C07321=1117.098,350.996,-84.045,-177.253,10.967,149.496
C07322=1117.094,351.244,-84.080,-177.250,10.969,149.496
C07323=1117.091,351.491,-84.116,-177.247,10.972,149.496
C07324=1117.087,351.738,-84.151,-177.243,10.974,149.496
C07325=1117.083,351.986,-84.186,-177.240,10.977,149.495
C07326=1117.078,352.233,-84.222,-177.236,10.979,149.495
C07327=1117.075,352.481,-84.258,-177.233,10.981,149.495
C07328=1117.071,352.729,-84.293,-177.230,10.984,149.495
C07329=1117.067,352.976,-84.328,-177.226,10.986,149.494
C07330=1117.063,353.223,-84.364,-177.222,10.989,149.494
C07331=1117.059,353.471,-84.399,-177.219,10.992,149.494
C07332=1117.056,353.718,-84.435,-177.216,10.994,149.494
C07333=1117.052,353.966,-84.470,-177.212,10.996,149.493
C07334=1117.048,354.213,-84.506,-177.209,10.999,149.493
C07335=1117.044,354.460,-84.541,-177.205,11.001,149.493
C07336=1117.040,354.708,-84.576,-177.202,11.004,149.493
C07337=1117.037,354.955,-84.612,-177.199,11.006,149.492
C07338=1117.032,355.203,-84.648,-177.196,11.009,149.492
C07339=1117.029,355.450,-84.684,-177.192,11.011,149.492
C07340=1117.025,355.698,-84.719,-177.188,11.013,149.492
C07341=1117.021,355.945,-84.755,-177.185,11.016,149.491
C07342=1117.017,356.192,-84.790,-177.182,11.018,149.491
C07343=1117.014,356.439,-84.826,-177.179,11.021,149.491
C07344=1117.009,356.687,-84.862,-177.175,11.023,149.491
C07345=1117.006,356.934,-84.898,-177.172,11.025,149.490
C07346=1117.002,357.182,-84.933,-177.168,11.028,149.490
C07347=1116.998,357.429,-84.969,-177.164,11.031,149.490
C07348=1116.995,357.677,-85.005,-177.161,11.033,149.490
C07349=1116.991,357.924,-85.041,-177.158,11.036,149.490
C07350=1116.987,358.172,-85.077,-177.154,11.038,149.489
C07351=1116.983,358.419,-85.113,-177.151,11.041,149.489
C07352=1116.980,358.667,-85.148,-177.147,11.043,149.489
C07353=1116.975,358.914,-85.185,-177.144,11.045,149.488
C07354=1116.972,359.161,-85.220,-177.141,11.048,149.488
C07355=1116.968,359.409,-85.256,-177.137,11.050,149.488
C07356=1116.963,359.656,-85.292,-177.134,11.053,149.488
C07357=1116.960,359.903,-85.328,-177.130,11.055,149.487
C07358=1116.956,360.150,-85.364,-177.127,11.057,149.487
C07359=1116.952,360.398,-85.400,-177.123,11.060,149.487
C07360=1116.948,360.645,-85.436,-177.120,11.062,149.487
C07361=1116.945,360.893,-85.472,-177.117,11.065,149.486
C07362=1116.941,361.140,-85.508,-177.114,11.067,149.486
C07363=1116.937,361.387,-85.544,-177.110,11.069,149.486
C07364=1116.934,361.600,-85.575,-177.108,11.071,149.486
C07365=1116.931,361.811,-85.606,-177.105,11.073,149.485
C07366=1116.927,362.023,-85.636,-177.102,11.075,149.485
C07367=1116.924,362.236,-85.668,-177.099,11.077,149.485
C07368=1116.921,362.447,-85.699,-177.096,11.079,149.485
C07369=1116.918,362.659,-85.730,-177.093,11.081,149.484
C07370=1116.915,362.872,-85.761,-177.090,11.083,149.484
C07371=1116.911,363.084,-85.792,-177.087,11.085,149.484
C07372=1116.907,363.331,-85.828,-177.084,11.088,149.484
C07373=1116.904,363.578,-85.864,-177.080,11.090,149.484
C07374=1116.900,363.825,-85.901,-177.077,11.093,149.483
C07375=1116.896,364.073,-85.937,-177.074,11.095,149.483
C07376=1116.893,364.321,-85.973,-177.070,11.097,149.483
C07377=1116.889,364.568,-86.009,-177.067,11.100,149.483
C07378=1116.885,364.815,-86.046,-177.063,11.102,149.482
C07379=1116.881,365.062,-86.083,-177.060,11.105,149.482
C07380=1116.878,365.310,-86.118,-177.057,11.106,149.482
C07381=1116.873,365.557,-86.155,-177.054,11.109,149.481
C07382=1116.870,365.804,-86.191,-177.050,11.111,149.481
C07383=1116.866,366.052,-86.227,-177.047,11.114,149.481
C07384=1116.862,366.299,-86.264,-177.044,11.116,149.481
C07385=1116.858,366.546,-86.301,-177.041,11.119,149.481
C07386=1116.854,366.794,-86.337,-177.037,11.121,149.480
C07387=1116.851,367.041,-86.373,-177.034,11.123,149.480
C07388=1116.847,367.288,-86.410,-177.030,11.126,149.480
C07389=1116.844,367.535,-86.446,-177.027,11.128,149.480
C07390=1116.840,367.783,-86.483,-177.024,11.131,149.479
C07391=1116.836,368.030,-86.519,-177.020,11.133,149.479
C07392=1116.832,368.277,-86.556,-177.017,11.136,149.479
C07393=1116.828,368.524,-86.593,-177.014,11.138,149.479
C07394=1116.825,368.772,-86.629,-177.010,11.140,149.478
C07395=1116.821,369.019,-86.666,-177.007,11.143,149.478
C07396=1116.817,369.266,-86.703,-177.003,11.145,149.478
C07397=1116.813,369.513,-86.739,-177.001,11.147,149.478
C07398=1116.809,369.761,-86.775,-176.997,11.149,149.477
C07399=1116.805,370.008,-86.812,-176.994,11.152,149.477
C07400=1116.802,370.256,-86.849,-176.991,11.154,149.477
C07401=1116.798,370.503,-86.886,-176.988,11.157,149.477
C07402=1116.794,370.750,-86.923,-176.984,11.159,149.477
C07403=1116.791,370.997,-86.959,-176.981,11.162,149.476
C07404=1116.787,371.244,-86.996,-176.978,11.164,149.476
C07405=1116.783,371.492,-87.033,-176.974,11.166,149.476
C07406=1116.779,371.739,-87.070,-176.971,11.169,149.476
C07407=1116.776,371.986,-87.106,-176.967,11.171,149.475
C07408=1116.771,372.233,-87.143,-176.964,11.174,149.475
C07409=1116.768,372.481,-87.181,-176.961,11.176,149.475
C07410=1116.764,372.728,-87.218,-176.957,11.179,149.475
C07411=1116.761,372.975,-87.254,-176.954,11.181,149.475
C07412=1116.757,373.222,-87.291,-176.952,11.183,149.474
C07413=1116.753,373.470,-87.328,-176.948,11.185,149.474
C07414=1116.749,373.717,-87.365,-176.945,11.188,149.474
C07415=1116.745,373.964,-87.402,-176.942,11.190,149.474
C07416=1116.742,374.212,-87.438,-176.939,11.193,149.474
C07417=1116.739,374.458,-87.476,-176.935,11.196,149.474
C07418=1116.734,374.706,-87.513,-176.932,11.198,149.473
C07419=1116.730,374.953,-87.550,-176.929,11.201,149.473
C07420=1116.728,375.165,-87.582,-176.926,11.202,149.473
C07421=1116.724,375.376,-87.613,-176.923,11.205,149.473
C07422=1116.721,375.589,-87.644,-176.921,11.207,149.473
C07423=1116.718,375.801,-87.677,-176.918,11.208,149.472
C07424=1116.714,376.012,-87.709,-176.915,11.211,149.472
C07425=1116.712,376.224,-87.741,-176.912,11.213,149.472
C07426=1116.708,376.436,-87.772,-176.909,11.215,149.472
C07427=1116.705,376.648,-87.805,-176.907,11.217,149.472
C07428=1116.702,376.895,-87.841,-176.903,11.220,149.472
C07429=1116.698,377.143,-87.878,-176.900,11.222,149.471
C07430=1116.694,377.389,-87.916,-176.897,11.225,149.471
C07431=1116.690,377.637,-87.953,-176.894,11.228,149.471
C07432=1116.687,377.885,-87.990,-176.891,11.230,149.471
C07433=1116.683,378.131,-88.028,-176.887,11.233,149.471
C07434=1116.679,378.378,-88.064,-176.884,11.235,149.471
C07435=1116.676,378.626,-88.102,-176.882,11.237,149.471
C07436=1116.671,378.873,-88.139,-176.879,11.240,149.470
C07437=1116.668,379.119,-88.177,-176.875,11.242,149.470
C07438=1116.664,379.367,-88.214,-176.872,11.245,149.470
C07439=1116.660,379.614,-88.252,-176.869,11.247,149.470
C07440=1116.657,379.862,-88.289,-176.866,11.250,149.470
C07441=1116.653,380.108,-88.326,-176.862,11.252,149.470
C07442=1116.649,380.355,-88.363,-176.860,11.255,149.470
C07443=1116.646,380.603,-88.401,-176.856,11.258,149.469
C07444=1116.642,380.850,-88.438,-176.853,11.260,149.469
C07445=1116.639,381.097,-88.476,-176.850,11.263,149.469
C07446=1116.634,381.345,-88.514,-176.847,11.266,149.469
C07447=1116.631,381.592,-88.551,-176.844,11.268,149.469
C07448=1116.627,381.839,-88.589,-176.841,11.271,149.469
C07449=1116.623,382.086,-88.626,-176.838,11.274,149.469
C07450=1116.619,382.333,-88.664,-176.834,11.276,149.469
C07451=1116.616,382.580,-88.701,-176.832,11.279,149.469
C07452=1116.612,382.827,-88.739,-176.828,11.281,149.468
C07453=1116.608,383.074,-88.776,-176.825,11.284,149.468
C07454=1116.605,383.321,-88.814,-176.822,11.287,149.468
C07455=1116.600,383.569,-88.852,-176.820,11.289,149.468
C07456=1116.597,383.816,-88.890,-176.817,11.292,149.468
C07457=1116.593,384.063,-88.927,-176.815,11.294,149.468
C07458=1116.590,384.310,-88.965,-176.813,11.296,149.468
C07459=1116.586,384.557,-89.002,-176.810,11.298,149.468
C07460=1116.583,384.804,-89.040,-176.808,11.301,149.468
C07461=1116.578,385.051,-89.078,-176.805,11.303,149.468
C07462=1116.575,385.299,-89.116,-176.803,11.305,149.468
C07463=1116.571,385.545,-89.154,-176.801,11.307,149.468
C07464=1116.568,385.792,-89.191,-176.799,11.310,149.468
C07465=1116.564,386.040,-89.228,-176.796,11.312,149.468
C07466=1116.560,386.287,-89.267,-176.795,11.315,149.468
C07467=1116.556,386.534,-89.304,-176.792,11.318,149.468
C07468=1116.553,386.781,-89.342,-176.790,11.320,149.469
C07469=1116.549,387.028,-89.380,-176.787,11.323,149.469
C07470=1116.546,387.275,-89.418,-176.785,11.325,149.469
C07471=1116.542,387.522,-89.456,-176.783,11.328,149.469
C07472=1116.539,387.769,-89.494,-176.780,11.330,149.469
C07473=1116.535,388.016,-89.532,-176.778,11.333,149.469
C07474=1116.531,388.263,-89.570,-176.776,11.336,149.469
C07475=1116.527,388.511,-89.607,-176.774,11.338,149.469
C07476=1116.525,388.722,-89.640,-176.772,11.341,149.469
C07477=1116.521,388.934,-89.672,-176.770,11.343,149.470
C07478=1116.518,389.145,-89.705,-176.768,11.345,149.470
C07479=1116.515,389.358,-89.738,-176.766,11.348,149.470
C07480=1116.513,389.569,-89.770,-176.765,11.350,149.470
C07481=1116.508,389.781,-89.802,-176.763,11.352,149.470
C07482=1116.505,389.993,-89.836,-176.761,11.355,149.470
C07483=1116.503,390.205,-89.868,-176.759,11.357,149.470
C07484=1116.499,390.452,-89.906,-176.756,11.360,149.471
C07485=1116.495,390.699,-89.944,-176.755,11.363,149.471
C07486=1116.492,390.946,-89.982,-176.752,11.366,149.471
C07487=1116.488,391.193,-90.019,-176.751,11.368,149.471
C07488=1116.484,391.440,-90.059,-176.748,11.372,149.471
C07489=1116.481,391.687,-90.097,-176.746,11.374,149.471
C07490=1116.477,391.933,-90.134,-176.744,11.377,149.472
C07491=1116.473,392.181,-90.173,-176.742,11.381,149.472
C07492=1116.470,392.428,-90.211,-176.740,11.383,149.472
C07493=1116.466,392.675,-90.249,-176.738,11.386,149.473
C07494=1116.462,392.922,-90.287,-176.736,11.390,149.473
C07495=1116.459,393.169,-90.326,-176.734,11.393,149.473
C07496=1116.455,393.416,-90.364,-176.732,11.396,149.473
C07497=1116.452,393.663,-90.401,-176.729,11.399,149.474
C07498=1116.447,393.910,-90.440,-176.728,11.402,149.474
C07499=1116.444,394.157,-90.478,-176.726,11.405,149.474
C07500=1116.440,394.404,-90.517,-176.724,11.409,149.475
C07501=1116.437,394.651,-90.554,-176.721,11.412,149.475
C07502=1116.433,394.898,-90.593,-176.720,11.415,149.475
C07503=1116.430,395.146,-90.631,-176.718,11.418,149.476
C07504=1116.426,395.393,-90.670,-176.716,11.422,149.476
C07505=1116.422,395.639,-90.708,-176.714,11.425,149.477
C07506=1116.418,395.887,-90.746,-176.712,11.429,149.477
C07507=1116.415,396.133,-90.785,-176.710,11.432,149.477
C07508=1116.411,396.380,-90.823,-176.708,11.435,149.478
C07509=1116.408,396.628,-90.861,-176.706,11.438,149.478
C07510=1116.404,396.875,-90.900,-176.704,11.442,149.479
C07511=1116.400,397.121,-90.938,-176.702,11.446,149.479
C07512=1116.397,397.368,-90.977,-176.700,11.450,149.480
C07513=1116.393,397.615,-91.015,-176.698,11.453,149.480
C07514=1116.390,397.863,-91.054,-176.697,11.457,149.480
C07515=1116.386,398.109,-91.092,-176.695,11.460,149.481
C07516=1116.382,398.356,-91.130,-176.693,11.464,149.481
C07517=1116.379,398.603,-91.169,-176.691,11.468,149.482
C07518=1116.375,398.851,-91.208,-176.689,11.471,149.482
C07519=1116.371,399.097,-91.246,-176.687,11.475,149.483
C07520=1116.368,399.344,-91.284,-176.686,11.479,149.483
C07521=1116.364,399.591,-91.324,-176.684,11.483,149.484
C07522=1116.361,399.838,-91.362,-176.682,11.487,149.485
C07523=1116.357,400.085,-91.400,-176.680,11.490,149.485
C07524=1116.353,400.332,-91.439,-176.679,11.494,149.486
C07525=1116.350,400.579,-91.478,-176.677,11.498,149.486
C07526=1116.346,400.827,-91.516,-176.675,11.502,149.487
C07527=1116.343,401.074,-91.555,-176.673,11.507,149.488
C07528=1116.339,401.319,-91.594,-176.672,11.510,149.488
C07529=1116.335,401.567,-91.632,-176.670,11.514,149.489
C07530=1116.331,401.814,-91.672,-176.669,11.518,149.489
C07531=1116.328,402.061,-91.709,-176.667,11.522,149.490
C07532=1116.325,402.273,-91.743,-176.665,11.526,149.491
C07533=1116.322,402.485,-91.776,-176.663,11.530,149.491
C07534=1116.319,402.696,-91.809,-176.663,11.533,149.492
C07535=1116.316,402.908,-91.843,-176.661,11.537,149.492
C07536=1116.314,403.119,-91.876,-176.659,11.541,149.493
C07537=1116.310,403.331,-91.909,-176.659,11.544,149.494
C07538=1116.307,403.542,-91.942,-176.657,11.548,149.494
C07539=1116.303,403.753,-91.976,-176.655,11.552,149.495
C07540=1116.300,404.000,-92.015,-176.654,11.556,149.495
C07541=1116.297,404.248,-92.053,-176.652,11.560,149.496
C07542=1116.293,404.495,-92.092,-176.650,11.565,149.497
C07543=1116.289,404.742,-92.131,-176.649,11.569,149.498
C07544=1116.286,404.988,-92.171,-176.647,11.574,149.499
C07545=1116.283,405.236,-92.209,-176.646,11.578,149.499
C07546=1116.279,405.483,-92.248,-176.645,11.582,149.500
C07547=1116.275,405.729,-92.287,-176.643,11.587,149.501
C07548=1116.271,405.976,-92.326,-176.642,11.592,149.502
C07549=1116.267,406.223,-92.365,-176.640,11.597,149.503
C07550=1116.265,406.470,-92.404,-176.639,11.601,149.503
C07551=1116.261,406.717,-92.442,-176.637,11.606,149.504
C07552=1116.257,406.964,-92.482,-176.636,11.610,149.505
C07553=1116.253,407.211,-92.521,-176.634,11.615,149.506
C07554=1116.250,407.458,-92.560,-176.633,11.620,149.507
C07555=1116.247,407.705,-92.599,-176.632,11.625,149.508
C07556=1116.243,407.952,-92.638,-176.630,11.630,149.509
C07557=1116.240,408.199,-92.677,-176.629,11.635,149.510
C07558=1116.236,408.446,-92.716,-176.628,11.640,149.511
C07559=1116.232,408.692,-92.755,-176.626,11.645,149.512
C07560=1116.228,408.939,-92.795,-176.625,11.649,149.513
C07561=1116.225,409.185,-92.833,-176.623,11.655,149.514
C07562=1116.222,409.432,-92.873,-176.622,11.660,149.515
C07563=1116.218,409.679,-92.912,-176.620,11.665,149.516
C07564=1116.214,409.926,-92.951,-176.620,11.670,149.517
C07565=1116.211,410.173,-92.990,-176.618,11.675,149.518
C07566=1116.207,410.420,-93.030,-176.617,11.681,149.519
C07567=1116.204,410.667,-93.069,-176.615,11.686,149.520
C07568=1116.200,410.914,-93.108,-176.614,11.691,149.521
C07569=1116.197,411.160,-93.148,-176.614,11.696,149.522
C07570=1116.193,411.407,-93.187,-176.612,11.701,149.523
C07571=1116.189,411.654,-93.227,-176.611,11.707,149.524
C07572=1116.186,411.901,-93.266,-176.610,11.713,149.525
C07573=1116.182,412.148,-93.305,-176.608,11.718,149.527
C07574=1116.179,412.395,-93.344,-176.607,11.724,149.528
C07575=1116.175,412.642,-93.384,-176.606,11.729,149.529
C07576=1116.172,412.889,-93.423,-176.605,11.735,149.530
C07577=1116.168,413.136,-93.463,-176.604,11.741,149.531
C07578=1116.164,413.382,-93.502,-176.603,11.746,149.533
C07579=1116.161,413.629,-93.541,-176.602,11.752,149.534
C07580=1116.159,413.876,-93.581,-176.601,11.758,149.535
C07581=1116.156,414.123,-93.620,-176.600,11.763,149.536
C07582=1116.154,414.370,-93.659,-176.599,11.769,149.537
C07583=1116.153,414.617,-93.699,-176.598,11.775,149.539
C07584=1116.152,414.864,-93.737,-176.597,11.780,149.540
C07585=1116.151,415.111,-93.777,-176.596,11.786,149.541
C07586=1116.151,415.358,-93.816,-176.595,11.792,149.543
C07587=1116.153,415.605,-93.854,-176.594,11.799,149.544
C07588=1116.154,415.816,-93.888,-176.593,11.804,149.545
C07589=1116.155,416.027,-93.922,-176.593,11.809,149.546
C07590=1116.156,416.239,-93.954,-176.592,11.814,149.548
C07591=1116.159,416.450,-93.988,-176.591,11.819,149.549
C07592=1116.161,416.661,-94.021,-176.590,11.825,149.550
C07593=1116.165,416.873,-94.054,-176.590,11.830,149.551
C07594=1116.168,417.084,-94.087,-176.589,11.835,149.552
C07595=1116.171,417.296,-94.120,-176.588,11.840,149.554
C07596=1115.753,417.296,-94.183,-176.581,11.845,149.553
C07597=1115.749,417.084,-94.150,-176.581,11.840,149.552
C07598=1115.745,416.872,-94.116,-176.582,11.834,149.550
C07599=1115.743,416.661,-94.084,-176.583,11.829,149.549
C07600=1115.740,416.450,-94.051,-176.584,11.824,149.548
C07601=1115.737,416.239,-94.017,-176.584,11.819,149.547
C07602=1115.736,416.027,-93.984,-176.586,11.813,149.546
C07603=1115.735,415.816,-93.951,-176.586,11.808,149.545
C07604=1115.734,415.605,-93.917,-176.587,11.802,149.543
C07605=1115.732,415.358,-93.878,-176.588,11.797,149.542
C07606=1115.732,415.111,-93.840,-176.589,11.791,149.541
C07607=1115.733,414.864,-93.800,-176.590,11.785,149.539
C07608=1115.734,414.617,-93.761,-176.591,11.779,149.538
C07609=1115.735,414.370,-93.722,-176.592,11.774,149.537
C07610=1115.737,414.123,-93.682,-176.593,11.767,149.536
C07611=1115.739,413.876,-93.643,-176.594,11.761,149.534
C07612=1115.743,413.629,-93.603,-176.595,11.756,149.533
C07613=1115.746,413.382,-93.565,-176.596,11.750,149.532
C07614=1115.750,413.135,-93.525,-176.597,11.744,149.531
C07615=1115.753,412.889,-93.485,-176.599,11.739,149.529
C07616=1115.757,412.642,-93.446,-176.600,11.733,149.528
C07617=1115.760,412.395,-93.406,-176.601,11.728,149.527
C07618=1115.764,412.148,-93.367,-176.602,11.722,149.526
C07619=1115.767,411.902,-93.328,-176.603,11.716,149.525
C07620=1115.770,411.655,-93.289,-176.605,11.711,149.524
C07621=1115.774,411.408,-93.249,-176.606,11.706,149.523
C07622=1115.777,411.161,-93.210,-176.607,11.700,149.522
C07623=1115.781,410.914,-93.171,-176.608,11.695,149.520
C07624=1115.785,410.667,-93.132,-176.610,11.689,149.519
C07625=1115.788,410.420,-93.092,-176.611,11.684,149.518
C07626=1115.792,410.174,-93.052,-176.613,11.679,149.517
C07627=1115.795,409.927,-93.013,-176.613,11.674,149.516
C07628=1115.799,409.680,-92.974,-176.615,11.669,149.515
C07629=1115.802,409.433,-92.935,-176.617,11.663,149.514
C07630=1115.806,409.186,-92.895,-176.618,11.658,149.513
C07631=1115.810,408.939,-92.856,-176.619,11.653,149.512
C07632=1115.813,408.692,-92.817,-176.620,11.648,149.511
C07633=1115.816,408.445,-92.778,-176.622,11.643,149.510
C07634=1115.820,408.198,-92.739,-176.623,11.638,149.509
C07635=1115.823,407.952,-92.700,-176.624,11.633,149.508
C07636=1115.827,407.705,-92.660,-176.626,11.628,149.508
C07637=1115.831,407.458,-92.621,-176.628,11.623,149.507
C07638=1115.834,407.211,-92.582,-176.629,11.619,149.506
C07639=1115.838,406.964,-92.543,-176.631,11.614,149.505
C07640=1115.841,406.717,-92.504,-176.632,11.609,149.504
C07641=1115.845,406.469,-92.465,-176.633,11.604,149.503
C07642=1115.848,406.222,-92.426,-176.635,11.599,149.502
C07643=1115.853,405.976,-92.387,-176.637,11.595,149.501
C07644=1115.856,405.729,-92.348,-176.638,11.590,149.500
C07645=1115.859,405.483,-92.309,-176.640,11.586,149.500
C07646=1115.863,405.236,-92.270,-176.642,11.581,149.499
C07647=1115.866,404.989,-92.231,-176.643,11.577,149.498
C07648=1115.870,404.741,-92.192,-176.645,11.572,149.497
C07649=1115.873,404.494,-92.154,-176.646,11.568,149.497
C07650=1115.877,404.247,-92.114,-176.648,11.563,149.496
C07651=1115.880,404.001,-92.075,-176.649,11.559,149.495
C07652=1115.885,403.754,-92.037,-176.651,11.554,149.494
C07653=1115.887,403.543,-92.004,-176.652,11.550,149.494
C07654=1115.890,403.331,-91.970,-176.654,11.547,149.493
C07655=1115.893,403.119,-91.937,-176.656,11.543,149.493
C07656=1115.897,402.908,-91.904,-176.657,11.540,149.492
C07657=1115.900,402.696,-91.870,-176.658,11.536,149.491
C07658=1115.903,402.484,-91.837,-176.660,11.532,149.491
C07659=1115.906,402.273,-91.804,-176.661,11.528,149.490
C07660=1115.908,402.061,-91.771,-176.663,11.525,149.490
C07661=1115.912,401.814,-91.732,-176.664,11.521,149.489
C07662=1115.916,401.567,-91.693,-176.666,11.516,149.488
C07663=1115.919,401.321,-91.655,-176.668,11.513,149.488
C07664=1115.923,401.074,-91.616,-176.670,11.509,149.487
C07665=1115.927,400.826,-91.577,-176.671,11.505,149.486
C07666=1115.930,400.580,-91.539,-176.673,11.500,149.486
C07667=1115.934,400.332,-91.500,-176.675,11.496,149.485
C07668=1115.938,400.086,-91.461,-176.677,11.492,149.485
C07669=1115.941,399.839,-91.423,-176.678,11.489,149.484
C07670=1115.945,399.591,-91.384,-176.680,11.485,149.484
C07671=1115.948,399.345,-91.345,-176.682,11.481,149.483
C07672=1115.952,399.098,-91.307,-176.684,11.477,149.483
C07673=1115.956,398.851,-91.268,-176.686,11.474,149.482
C07674=1115.959,398.604,-91.230,-176.687,11.470,149.482
C07675=1115.963,398.357,-91.191,-176.689,11.466,149.481
C07676=1115.966,398.110,-91.153,-176.691,11.463,149.481
C07677=1115.970,397.863,-91.115,-176.694,11.458,149.480
C07678=1115.973,397.616,-91.076,-176.696,11.455,149.480
C07679=1115.977,397.368,-91.037,-176.697,11.452,149.479
C07680=1115.981,397.122,-90.999,-176.699,11.448,149.479
C07681=1115.985,396.875,-90.961,-176.701,11.444,149.478
C07682=1115.989,396.627,-90.922,-176.703,11.441,149.478
C07683=1115.991,396.381,-90.883,-176.705,11.437,149.478
C07684=1115.996,396.134,-90.845,-176.707,11.434,149.477
C07685=1115.999,395.887,-90.807,-176.709,11.430,149.477
C07686=1116.003,395.639,-90.768,-176.711,11.427,149.476
C07687=1116.007,395.393,-90.730,-176.713,11.423,149.476
C07688=1116.010,395.145,-90.692,-176.715,11.420,149.476
C07689=1116.013,394.899,-90.653,-176.717,11.416,149.475
C07690=1116.018,394.652,-90.615,-176.719,11.414,149.475
C07691=1116.021,394.404,-90.577,-176.721,11.410,149.474
C07692=1116.025,394.158,-90.538,-176.723,11.407,149.474
C07693=1116.028,393.911,-90.500,-176.725,11.404,149.474
C07694=1116.032,393.664,-90.462,-176.727,11.401,149.474
C07695=1116.036,393.416,-90.424,-176.729,11.397,149.473
C07696=1116.039,393.170,-90.386,-176.731,11.394,149.473
C07697=1116.043,392.923,-90.347,-176.733,11.391,149.473
C07698=1116.046,392.675,-90.309,-176.735,11.388,149.472
C07699=1116.051,392.428,-90.271,-176.737,11.385,149.472
C07700=1116.054,392.181,-90.233,-176.740,11.381,149.472
C07701=1116.057,391.934,-90.195,-176.741,11.379,149.472
C07702=1116.062,391.687,-90.157,-176.744,11.376,149.471
C07703=1116.064,391.440,-90.118,-176.746,11.372,149.471
C07704=1116.068,391.193,-90.080,-176.748,11.370,149.471
C07705=1116.072,390.946,-90.042,-176.750,11.367,149.471
C07706=1116.075,390.699,-90.004,-176.753,11.364,149.471
C07707=1116.079,390.452,-89.967,-176.754,11.361,149.470
C07708=1116.083,390.205,-89.928,-176.757,11.358,149.470
C07709=1116.086,389.993,-89.895,-176.759,11.356,149.470
C07710=1116.089,389.781,-89.863,-176.761,11.353,149.470
C07711=1116.092,389.570,-89.830,-176.763,11.351,149.470
C07712=1116.096,389.358,-89.798,-176.764,11.349,149.470
C07713=1116.098,389.146,-89.766,-176.766,11.346,149.469
C07714=1116.101,388.934,-89.733,-176.768,11.344,149.469
C07715=1116.105,388.723,-89.701,-176.770,11.341,149.469
C07716=1116.108,388.511,-89.668,-176.772,11.339,149.469
C07717=1116.111,388.264,-89.630,-176.774,11.337,149.469
C07718=1116.116,388.017,-89.592,-176.777,11.334,149.469
C07719=1116.119,387.770,-89.554,-176.779,11.332,149.469
C07720=1116.123,387.523,-89.516,-176.781,11.328,149.469
C07721=1116.126,387.276,-89.478,-176.783,11.326,149.469
C07722=1116.131,387.028,-89.441,-176.786,11.323,149.468
C07723=1116.134,386.781,-89.403,-176.788,11.321,149.468
C07724=1116.137,386.534,-89.365,-176.791,11.318,149.468
C07725=1116.141,386.287,-89.327,-176.792,11.316,149.468
C07726=1116.144,386.040,-89.289,-176.795,11.314,149.468
C07727=1116.149,385.793,-89.251,-176.797,11.311,149.468
C07728=1116.152,385.546,-89.213,-176.800,11.309,149.468
C07729=1116.156,385.299,-89.176,-176.802,11.306,149.468
C07730=1116.159,385.051,-89.138,-176.804,11.303,149.468
C07731=1116.163,384.805,-89.101,-176.807,11.301,149.468
C07732=1116.167,384.557,-89.062,-176.809,11.299,149.468
C07733=1116.170,384.311,-89.025,-176.812,11.296,149.468
C07734=1116.174,384.063,-88.987,-176.814,11.294,149.468
C07735=1116.178,383.816,-88.950,-176.816,11.292,149.468
C07736=1116.181,383.569,-88.912,-176.818,11.290,149.468
C07737=1116.185,383.322,-88.874,-176.821,11.287,149.468
C07738=1116.189,383.074,-88.837,-176.824,11.285,149.468
C07739=1116.193,382.828,-88.799,-176.827,11.282,149.468
C07740=1116.196,382.580,-88.761,-176.831,11.279,149.468
C07741=1116.200,382.333,-88.724,-176.833,11.277,149.468
C07742=1116.203,382.086,-88.686,-176.837,11.274,149.469
C07743=1116.207,381.839,-88.649,-176.840,11.271,149.469
C07744=1116.211,381.592,-88.612,-176.843,11.269,149.469
C07745=1116.214,381.345,-88.574,-176.846,11.266,149.469
C07746=1116.218,381.098,-88.536,-176.849,11.264,149.469
C07747=1116.222,380.850,-88.499,-176.852,11.261,149.469
C07748=1116.226,380.604,-88.461,-176.855,11.258,149.469
C07749=1116.230,380.356,-88.424,-176.859,11.256,149.469
C07750=1116.233,380.109,-88.386,-176.862,11.253,149.470
C07751=1116.237,379.862,-88.349,-176.865,11.250,149.470
C07752=1116.241,379.615,-88.311,-176.868,11.248,149.470
C07753=1116.245,379.367,-88.274,-176.871,11.245,149.470
C07754=1116.248,379.120,-88.236,-176.874,11.243,149.470
C07755=1116.252,378.873,-88.200,-176.878,11.240,149.470
C07756=1116.256,378.626,-88.162,-176.881,11.238,149.470
C07757=1116.259,378.379,-88.125,-176.884,11.235,149.471
C07758=1116.263,378.132,-88.087,-176.887,11.232,149.471
C07759=1116.267,377.885,-88.050,-176.890,11.231,149.471
C07760=1116.270,377.638,-88.012,-176.893,11.228,149.471
C07761=1116.274,377.390,-87.976,-176.896,11.226,149.471
C07762=1116.279,377.143,-87.939,-176.900,11.223,149.472
C07763=1116.281,376.896,-87.901,-176.902,11.220,149.472
C07764=1116.285,376.649,-87.865,-176.906,11.218,149.472
C07765=1116.289,376.437,-87.832,-176.909,11.215,149.472
C07766=1116.292,376.225,-87.800,-176.911,11.213,149.472
C07767=1116.295,376.013,-87.769,-176.914,11.212,149.472
C07768=1116.298,375.801,-87.737,-176.917,11.209,149.472
C07769=1116.301,375.589,-87.705,-176.920,11.207,149.472
C07770=1116.305,375.378,-87.673,-176.923,11.205,149.473
C07771=1116.308,375.166,-87.641,-176.926,11.203,149.473
C07772=1116.311,374.954,-87.609,-176.928,11.201,149.473
C07773=1116.315,374.706,-87.572,-176.931,11.199,149.473
C07774=1116.319,374.459,-87.536,-176.934,11.196,149.473
C07775=1116.322,374.212,-87.499,-176.938,11.194,149.474
C07776=1116.326,373.964,-87.462,-176.941,11.191,149.474
C07777=1116.330,373.717,-87.425,-176.944,11.189,149.474
C07778=1116.334,373.471,-87.388,-176.948,11.186,149.474
C07779=1116.338,373.224,-87.351,-176.951,11.184,149.474
C07780=1116.340,372.976,-87.314,-176.954,11.181,149.475
C07781=1116.344,372.729,-87.277,-176.957,11.179,149.475
C07782=1116.349,372.482,-87.240,-176.961,11.176,149.475
C07783=1116.353,372.234,-87.204,-176.964,11.174,149.475
C07784=1116.355,371.987,-87.167,-176.967,11.171,149.475
C07785=1116.360,371.740,-87.130,-176.970,11.170,149.476
C07786=1116.364,371.492,-87.093,-176.973,11.167,149.476
C07787=1116.368,371.245,-87.056,-176.977,11.165,149.476
C07788=1116.370,370.998,-87.020,-176.980,11.162,149.476
C07789=1116.375,370.750,-86.983,-176.983,11.160,149.477
C07790=1116.379,370.503,-86.946,-176.987,11.157,149.477
C07791=1116.383,370.256,-86.909,-176.990,11.155,149.477
C07792=1116.386,370.009,-86.873,-176.993,11.152,149.477
C07793=1116.390,369.761,-86.836,-176.997,11.150,149.478
C07794=1116.394,369.514,-86.799,-177.000,11.148,149.478
C07795=1116.397,369.267,-86.763,-177.003,11.145,149.478
C07796=1116.401,369.020,-86.726,-177.007,11.143,149.478
C07797=1116.405,368.773,-86.689,-177.010,11.140,149.478
C07798=1116.408,368.525,-86.652,-177.013,11.138,149.479
C07799=1116.412,368.277,-86.616,-177.017,11.135,149.479
C07800=1116.416,368.031,-86.580,-177.020,11.133,149.479
C07801=1116.420,367.783,-86.543,-177.024,11.131,149.479
C07802=1116.424,367.536,-86.506,-177.026,11.129,149.480
C07803=1116.427,367.289,-86.470,-177.030,11.126,149.480
C07804=1116.432,367.042,-86.434,-177.033,11.124,149.480
C07805=1116.435,366.795,-86.397,-177.036,11.121,149.480
C07806=1116.439,366.547,-86.360,-177.040,11.119,149.480
C07807=1116.442,366.300,-86.324,-177.043,11.116,149.481
C07808=1116.446,366.052,-86.288,-177.047,11.114,149.481
C07809=1116.450,365.805,-86.251,-177.050,11.112,149.481
C07810=1116.454,365.558,-86.215,-177.053,11.109,149.481
C07811=1116.458,365.310,-86.178,-177.056,11.107,149.482
C07812=1116.462,365.063,-86.142,-177.060,11.104,149.482
C07813=1116.466,364.816,-86.105,-177.063,11.102,149.482
C07814=1116.469,364.569,-86.070,-177.067,11.100,149.483
C07815=1116.473,364.321,-86.033,-177.070,11.097,149.483
C07816=1116.477,364.075,-85.997,-177.073,11.095,149.483
C07817=1116.481,363.826,-85.960,-177.077,11.092,149.483
C07818=1116.484,363.579,-85.924,-177.080,11.090,149.484
C07819=1116.488,363.332,-85.888,-177.084,11.088,149.484
C07820=1116.492,363.084,-85.852,-177.087,11.085,149.484
C07821=1116.495,362.873,-85.821,-177.090,11.084,149.484
C07822=1116.498,362.661,-85.790,-177.092,11.082,149.484
C07823=1116.501,362.448,-85.759,-177.096,11.079,149.485
C07824=1116.505,362.236,-85.728,-177.098,11.078,149.485
C07825=1116.509,362.024,-85.697,-177.101,11.075,149.485
C07826=1116.511,361.813,-85.666,-177.104,11.073,149.485
C07827=1116.514,361.601,-85.635,-177.107,11.072,149.486
C07828=1116.518,361.389,-85.604,-177.110,11.069,149.486
C07829=1116.521,361.141,-85.568,-177.113,11.067,149.486
C07830=1116.526,360.894,-85.532,-177.117,11.065,149.486
C07831=1116.529,360.647,-85.496,-177.120,11.062,149.487
C07832=1116.533,360.399,-85.460,-177.123,11.060,149.487
C07833=1116.537,360.152,-85.424,-177.127,11.057,149.487
C07834=1116.541,359.904,-85.388,-177.130,11.055,149.487
C07835=1116.544,359.657,-85.353,-177.134,11.053,149.488
C07836=1116.548,359.410,-85.316,-177.137,11.050,149.488
C07837=1116.552,359.162,-85.280,-177.140,11.048,149.488
C07838=1116.556,358.915,-85.245,-177.144,11.045,149.488
C07839=1116.559,358.668,-85.208,-177.147,11.043,149.489
C07840=1116.563,358.420,-85.172,-177.151,11.041,149.489
C07841=1116.567,358.172,-85.137,-177.154,11.038,149.489
C07842=1116.571,357.925,-85.101,-177.157,11.036,149.489
C07843=1116.574,357.678,-85.065,-177.161,11.033,149.490
C07844=1116.579,357.430,-85.029,-177.164,11.031,149.490
C07845=1116.582,357.183,-84.993,-177.168,11.029,149.490
C07846=1116.586,356.935,-84.958,-177.171,11.026,149.490
C07847=1116.590,356.688,-84.922,-177.174,11.024,149.491
C07848=1116.594,356.441,-84.887,-177.178,11.021,149.491
C07849=1116.598,356.193,-84.851,-177.181,11.019,149.491
C07850=1116.602,355.946,-84.814,-177.185,11.017,149.491
C07851=1116.605,355.699,-84.779,-177.188,11.014,149.492
C07852=1116.609,355.451,-84.743,-177.191,11.012,149.492
C07853=1116.613,355.204,-84.708,-177.194,11.009,149.492
C07854=1116.616,354.956,-84.672,-177.198,11.007,149.492
C07855=1116.620,354.709,-84.637,-177.201,11.005,149.493
C07856=1116.625,354.462,-84.601,-177.205,11.002,149.493
C07857=1116.629,354.214,-84.565,-177.209,10.999,149.493
C07858=1116.632,353.967,-84.530,-177.212,10.996,149.493
C07859=1116.636,353.719,-84.494,-177.215,10.994,149.494
C07860=1116.640,353.472,-84.459,-177.219,10.991,149.494
C07861=1116.643,353.224,-84.423,-177.222,10.989,149.494
C07862=1116.647,352.977,-84.388,-177.226,10.987,149.494
C07863=1116.651,352.730,-84.352,-177.229,10.984,149.495
C07864=1116.655,352.482,-84.318,-177.232,10.982,149.495
C07865=1116.659,352.234,-84.282,-177.236,10.979,149.495
C07866=1116.662,351.987,-84.247,-177.239,10.977,149.495
C07867=1116.667,351.740,-84.211,-177.242,10.974,149.496
C07868=1116.670,351.492,-84.176,-177.246,10.971,149.496
C07869=1116.674,351.245,-84.140,-177.249,10.969,149.496
C07870=1116.678,350.997,-84.105,-177.253,10.966,149.496
C07871=1116.682,350.749,-84.070,-177.256,10.964,149.496
C07872=1116.686,350.503,-84.035,-177.260,10.962,149.497
C07873=1116.690,350.255,-83.999,-177.263,10.959,149.497
C07874=1116.694,350.007,-83.964,-177.266,10.957,149.497
C07875=1116.698,349.760,-83.929,-177.270,10.954,149.498
C07876=1116.701,349.513,-83.894,-177.274,10.951,149.498
C07877=1116.705,349.300,-83.863,-177.276,10.949,149.498
C07878=1116.708,349.088,-83.833,-177.279,10.947,149.498
C07879=1116.712,348.876,-83.803,-177.282,10.945,149.498
C07880=1116.715,348.664,-83.772,-177.284,10.943,149.498
C07881=1116.718,348.451,-83.743,-177.287,10.941,149.499
C07882=1116.722,348.239,-83.712,-177.290,10.938,149.499
C07883=1116.725,348.027,-83.682,-177.293,10.937,149.499
C07884=1116.728,347.815,-83.652,-177.295,10.935,149.499
C07885=1116.732,347.567,-83.617,-177.298,10.932,149.499
C07886=1116.736,347.320,-83.582,-177.301,10.930,149.499
C07887=1116.740,347.072,-83.547,-177.305,10.927,149.500
C07888=1116.744,346.824,-83.512,-177.308,10.925,149.500
C07889=1116.748,346.577,-83.477,-177.311,10.922,149.500
C07890=1116.751,346.330,-83.443,-177.314,10.920,149.500
C07891=1116.755,346.082,-83.407,-177.318,10.917,149.500
C07892=1116.759,345.835,-83.373,-177.321,10.915,149.501
C07893=1116.763,345.587,-83.337,-177.324,10.912,149.501
C07894=1116.768,345.340,-83.303,-177.328,10.910,149.501
C07895=1116.771,345.092,-83.267,-177.331,10.907,149.501
C07896=1116.775,344.845,-83.233,-177.334,10.905,149.501
C07897=1116.779,344.598,-83.198,-177.336,10.903,149.502
C07898=1116.783,344.350,-83.163,-177.340,10.900,149.502
C07899=1116.787,344.101,-83.128,-177.343,10.898,149.502
C07900=1116.790,343.855,-83.093,-177.346,10.896,149.502
C07901=1116.794,343.607,-83.059,-177.349,10.893,149.502
C07902=1116.799,343.359,-83.024,-177.353,10.890,149.503
C07903=1116.803,343.112,-82.989,-177.356,10.888,149.503
C07904=1116.806,342.865,-82.955,-177.359,10.885,149.503
C07905=1116.810,342.617,-82.920,-177.363,10.883,149.503
C07906=1116.814,342.369,-82.884,-177.365,10.880,149.503
C07907=1116.819,342.122,-82.850,-177.369,10.878,149.504
C07908=1116.822,341.874,-82.816,-177.372,10.875,149.504
C07909=1116.826,341.627,-82.781,-177.375,10.874,149.504
C07910=1116.830,341.379,-82.746,-177.378,10.871,149.504
C07911=1116.834,341.132,-82.712,-177.381,10.868,149.504
C07912=1116.838,340.884,-82.677,-177.384,10.866,149.505
C07913=1116.842,340.636,-82.642,-177.388,10.863,149.505
C07914=1116.846,340.389,-82.608,-177.391,10.861,149.505
C07915=1116.850,340.142,-82.573,-177.394,10.858,149.505
C07916=1116.853,339.894,-82.539,-177.397,10.856,149.505
C07917=1116.858,339.647,-82.504,-177.401,10.853,149.506
C07918=1116.862,339.398,-82.469,-177.404,10.851,149.506
C07919=1116.865,339.151,-82.436,-177.407,10.848,149.506
C07920=1116.869,338.903,-82.401,-177.410,10.846,149.506
C07921=1116.874,338.656,-82.366,-177.413,10.843,149.506
C07922=1116.877,338.408,-82.332,-177.416,10.841,149.507
C07923=1116.882,338.161,-82.298,-177.419,10.839,149.507
C07924=1116.885,337.913,-82.263,-177.423,10.837,149.507
C07925=1116.890,337.665,-82.229,-177.426,10.834,149.507
C07926=1116.893,337.418,-82.195,-177.429,10.831,149.507
C07927=1116.897,337.170,-82.160,-177.432,10.829,149.508
C07928=1116.901,336.922,-82.126,-177.436,10.826,149.508
C07929=1116.905,336.675,-82.091,-177.438,10.824,149.508
C07930=1116.908,336.427,-82.057,-177.442,10.821,149.508
C07931=1116.913,336.180,-82.023,-177.445,10.819,149.508
C07932=1116.916,335.932,-81.989,-177.448,10.816,149.509
C07933=1116.920,335.720,-81.959,-177.451,10.814,149.509
C07934=1116.923,335.508,-81.930,-177.453,10.813,149.509
C07935=1116.927,335.295,-81.901,-177.456,10.810,149.509
C07936=1116.930,335.083,-81.871,-177.459,10.808,149.509
C07937=1116.933,334.871,-81.842,-177.461,10.806,149.509
C07938=1116.937,334.658,-81.813,-177.465,10.804,149.510
C07939=1116.940,334.446,-81.783,-177.467,10.802,149.510
C07940=1116.944,334.234,-81.754,-177.470,10.799,149.510
C07941=1116.947,333.986,-81.720,-177.473,10.797,149.510
C07942=1116.952,333.738,-81.686,-177.476,10.795,149.510
C07943=1116.955,333.490,-81.652,-177.479,10.792,149.510
C07944=1116.959,333.243,-81.618,-177.482,10.789,149.511
C07945=1116.964,332.996,-81.583,-177.485,10.787,149.511
C07946=1116.967,332.747,-81.550,-177.489,10.785,149.511
C07947=1116.971,332.500,-81.516,-177.492,10.782,149.511
C07948=1116.975,332.253,-81.482,-177.495,10.779,149.511
C07949=1116.979,332.005,-81.447,-177.498,10.777,149.512
C07950=1116.983,331.757,-81.414,-177.502,10.774,149.512
C07951=1116.987,331.510,-81.380,-177.505,10.772,149.512
C07952=1116.991,331.262,-81.345,-177.508,10.769,149.512
C07953=1116.995,331.014,-81.312,-177.511,10.768,149.512
C07954=1116.999,330.767,-81.278,-177.514,10.765,149.513
C07955=1117.003,330.518,-81.244,-177.517,10.762,149.513
C07956=1117.007,330.271,-81.210,-177.520,10.760,149.513
C07957=1117.011,330.024,-81.177,-177.523,10.757,149.513
C07958=1117.015,329.776,-81.142,-177.526,10.755,149.513
C07959=1117.019,329.528,-81.109,-177.530,10.752,149.513
C07960=1117.023,329.281,-81.075,-177.533,10.750,149.514
C07961=1117.026,329.033,-81.041,-177.536,10.747,149.514
C07962=1117.031,328.785,-81.007,-177.539,10.745,149.514
C07963=1117.035,328.538,-80.974,-177.543,10.742,149.514
C07964=1117.039,328.290,-80.940,-177.546,10.740,149.514
C07965=1117.042,328.042,-80.906,-177.549,10.737,149.515
C07966=1117.046,327.794,-80.873,-177.551,10.735,149.515
C07967=1117.051,327.547,-80.839,-177.555,10.733,149.515
C07968=1117.055,327.299,-80.805,-177.558,10.730,149.515
C07969=1117.058,327.051,-80.772,-177.561,10.727,149.515
C07970=1117.062,326.804,-80.738,-177.564,10.725,149.516
C07971=1117.066,326.556,-80.705,-177.567,10.722,149.516
C07972=1117.070,326.309,-80.671,-177.571,10.720,149.516
C07973=1117.074,326.061,-80.637,-177.574,10.717,149.516
C07974=1117.079,325.812,-80.604,-177.577,10.715,149.516
C07975=1117.083,325.565,-80.570,-177.580,10.712,149.516
C07976=1117.087,325.318,-80.537,-177.583,10.710,149.517
C07977=1117.091,325.070,-80.503,-177.586,10.707,149.517
C07978=1117.094,324.821,-80.470,-177.589,10.705,149.517
C07979=1117.098,324.574,-80.436,-177.592,10.703,149.517
C07980=1117.102,324.327,-80.403,-177.595,10.700,149.517
C07981=1117.106,324.079,-80.370,-177.599,10.698,149.518
C07982=1117.111,323.831,-80.337,-177.602,10.695,149.518
C07983=1117.114,323.583,-80.302,-177.605,10.692,149.518
C07984=1117.118,323.336,-80.269,-177.608,10.690,149.518
C07985=1117.122,323.088,-80.236,-177.612,10.687,149.518
C07986=1117.126,322.840,-80.203,-177.614,10.685,149.518
C07987=1117.130,322.592,-80.170,-177.618,10.682,149.519
C07988=1117.134,322.345,-80.136,-177.621,10.679,149.519
C07989=1117.138,322.132,-80.107,-177.623,10.678,149.519
C07990=1117.140,321.920,-80.079,-177.626,10.676,149.519
C07991=1117.145,321.708,-80.050,-177.629,10.673,149.519
C07992=1117.147,321.495,-80.022,-177.631,10.671,149.519
C07993=1117.151,321.282,-79.993,-177.634,10.669,149.520
C07994=1117.154,321.070,-79.965,-177.637,10.667,149.520
C07995=1117.158,320.858,-79.936,-177.639,10.665,149.520
C07996=1117.161,320.646,-79.908,-177.642,10.663,149.520
C07997=1117.165,320.397,-79.875,-177.645,10.660,149.520
C07998=1117.169,320.150,-79.842,-177.648,10.658,149.521
C07999=1117.173,319.902,-79.808,-177.652,10.656,149.521
C08000=1117.177,319.654,-79.775,-177.654,10.653,149.521
C08001=1117.181,319.406,-79.742,-177.658,10.650,149.521
C08002=1117.185,319.159,-79.709,-177.661,10.648,149.521
C08003=1117.190,318.911,-79.676,-177.664,10.645,149.521
C08004=1117.193,318.663,-79.643,-177.667,10.643,149.522
C08005=1117.197,318.415,-79.611,-177.670,10.640,149.522
C08006=1117.202,318.167,-79.578,-177.674,10.637,149.522
C08007=1117.206,317.920,-79.545,-177.677,10.635,149.522
C08008=1117.210,317.672,-79.511,-177.679,10.633,149.522
C08009=1117.213,317.424,-79.478,-177.683,10.631,149.523
C08010=1117.217,317.176,-79.445,-177.685,10.628,149.523
C08011=1117.221,316.928,-79.412,-177.689,10.625,149.523
C08012=1117.225,316.680,-79.380,-177.692,10.623,149.523
C08013=1117.229,316.432,-79.347,-177.695,10.620,149.523
C08014=1117.233,316.185,-79.314,-177.698,10.618,149.523
C08015=1117.237,315.937,-79.281,-177.701,10.615,149.524
C08016=1117.241,315.689,-79.248,-177.705,10.613,149.524
C08017=1117.246,315.441,-79.215,-177.708,10.610,149.524
C08018=1117.249,315.194,-79.183,-177.711,10.607,149.524
C08019=1117.253,314.946,-79.149,-177.714,10.606,149.524
C08020=1117.258,314.698,-79.117,-177.716,10.603,149.524
C08021=1117.261,314.450,-79.084,-177.720,10.600,149.525
C08022=1117.265,314.202,-79.051,-177.723,10.598,149.525
C08023=1117.269,313.955,-79.018,-177.726,10.595,149.525
C08024=1117.273,313.707,-78.986,-177.729,10.593,149.525
C08025=1117.278,313.460,-78.954,-177.732,10.590,149.525
C08026=1117.282,313.211,-78.921,-177.736,10.588,149.526
C08027=1117.286,312.964,-78.889,-177.739,10.585,149.526
C08028=1117.290,312.716,-78.855,-177.742,10.582,149.526
C08029=1117.294,312.468,-78.823,-177.745,10.580,149.526
C08030=1117.298,312.220,-78.790,-177.748,10.577,149.526
C08031=1117.302,311.972,-78.758,-177.751,10.575,149.527
C08032=1117.306,311.724,-78.725,-177.754,10.573,149.527
C08033=1117.310,311.476,-78.693,-177.757,10.570,149.527
C08034=1117.314,311.228,-78.660,-177.760,10.568,149.527
C08035=1117.318,310.980,-78.628,-177.763,10.565,149.527
C08036=1117.322,310.733,-78.595,-177.767,10.563,149.527
C08037=1117.326,310.484,-78.562,-177.770,10.560,149.528
C08038=1117.330,310.238,-78.530,-177.773,10.557,149.528
C08039=1117.335,309.989,-78.498,-177.776,10.555,149.528
C08040=1117.338,309.742,-78.465,-177.779,10.552,149.528
C08041=1117.343,309.494,-78.433,-177.782,10.549,149.528
C08042=1117.346,309.245,-78.401,-177.785,10.548,149.529
C08043=1117.350,308.998,-78.368,-177.788,10.545,149.529
C08044=1117.354,308.750,-78.336,-177.791,10.543,149.529
C08045=1117.358,308.537,-78.309,-177.794,10.540,149.529
C08046=1117.362,308.325,-78.280,-177.797,10.538,149.529
C08047=1117.365,308.112,-78.253,-177.799,10.536,149.529
C08048=1117.369,307.899,-78.225,-177.802,10.533,149.529
C08049=1117.371,307.687,-78.197,-177.805,10.532,149.530
C08050=1117.375,307.474,-78.170,-177.807,10.530,149.530
C08051=1117.380,307.262,-78.142,-177.810,10.527,149.530
C08052=1117.382,307.049,-78.114,-177.813,10.525,149.530
C08053=1117.386,306.801,-78.082,-177.816,10.523,149.530
C08054=1117.391,306.553,-78.050,-177.819,10.520,149.530
C08055=1117.395,306.305,-78.018,-177.822,10.517,149.531
C08056=1117.399,306.058,-77.985,-177.825,10.515,149.531
C08057=1117.403,305.809,-77.953,-177.828,10.512,149.531
C08058=1117.407,305.562,-77.922,-177.831,10.510,149.531
C08059=1117.411,305.314,-77.889,-177.834,10.508,149.531
C08060=1117.415,305.066,-77.857,-177.837,10.505,149.532
C08061=1117.419,304.818,-77.825,-177.840,10.502,149.532
C08062=1117.424,304.571,-77.793,-177.843,10.500,149.532
C08063=1117.427,304.323,-77.761,-177.847,10.498,149.532
C08064=1117.432,304.074,-77.728,-177.850,10.495,149.532
C08065=1117.435,303.826,-77.696,-177.853,10.492,149.532
C08066=1117.440,303.579,-77.665,-177.856,10.490,149.533
C08067=1117.444,303.331,-77.633,-177.859,10.487,149.533
C08068=1117.448,303.083,-77.601,-177.862,10.484,149.533
C08069=1117.452,302.835,-77.569,-177.865,10.482,149.533
C08070=1117.457,302.587,-77.537,-177.868,10.480,149.533
C08071=1117.460,302.339,-77.505,-177.871,10.478,149.534
C08072=1117.464,302.091,-77.473,-177.874,10.475,149.534
C08073=1117.468,301.843,-77.442,-177.877,10.472,149.534
C08074=1117.473,301.595,-77.409,-177.880,10.470,149.534
C08075=1117.477,301.347,-77.377,-177.884,10.467,149.534
C08076=1117.481,301.100,-77.346,-177.886,10.464,149.534
C08077=1117.485,300.852,-77.314,-177.890,10.462,149.535
C08078=1117.489,300.603,-77.282,-177.893,10.459,149.535
C08079=1117.493,300.356,-77.250,-177.896,10.457,149.535
C08080=1117.497,300.107,-77.219,-177.898,10.455,149.535
C08081=1117.501,299.859,-77.187,-177.902,10.452,149.535
C08082=1117.505,299.612,-77.156,-177.905,10.450,149.535
C08083=1117.510,299.364,-77.123,-177.908,10.447,149.536
C08084=1117.513,299.116,-77.091,-177.911,10.444,149.536
C08085=1117.518,298.868,-77.060,-177.914,10.442,149.536
C08086=1117.522,298.620,-77.029,-177.917,10.439,149.536
C08087=1117.525,298.372,-76.997,-177.921,10.437,149.536
C08088=1117.530,298.124,-76.965,-177.923,10.434,149.536
C08089=1117.533,297.876,-76.934,-177.927,10.432,149.537
C08090=1117.539,297.628,-76.902,-177.929,10.430,149.537
C08091=1117.543,297.380,-76.870,-177.932,10.427,149.537
C08092=1117.546,297.132,-76.839,-177.935,10.424,149.537
C08093=1117.551,296.884,-76.807,-177.939,10.422,149.537
C08094=1117.555,296.636,-76.776,-177.942,10.419,149.537
C08095=1117.559,296.388,-76.744,-177.945,10.417,149.538
C08096=1117.563,296.140,-76.713,-177.948,10.414,149.538
C08097=1117.567,295.892,-76.682,-177.951,10.412,149.538
C08098=1117.571,295.644,-76.650,-177.954,10.409,149.538
C08099=1117.575,295.396,-76.619,-177.957,10.406,149.538
C08100=1117.579,295.148,-76.587,-177.960,10.404,149.539
C08101=1117.583,294.936,-76.560,-177.963,10.402,149.539
C08102=1117.586,294.722,-76.533,-177.965,10.400,149.539
C08103=1117.590,294.510,-76.506,-177.968,10.397,149.539
C08104=1117.593,294.298,-76.479,-177.971,10.395,149.539
C08105=1117.597,294.084,-76.453,-177.973,10.393,149.539
C08106=1117.601,293.872,-76.426,-177.976,10.391,149.540
C08107=1117.604,293.659,-76.398,-177.979,10.389,149.540
C08108=1117.607,293.446,-76.372,-177.981,10.387,149.540
C08109=1117.611,293.199,-76.341,-177.984,10.384,149.540
C08110=1117.615,292.950,-76.310,-177.987,10.382,149.540
C08111=1117.620,292.703,-76.278,-177.991,10.379,149.540
C08112=1117.624,292.454,-76.247,-177.993,10.376,149.540
C08113=1117.628,292.206,-76.216,-177.996,10.374,149.541
C08114=1117.632,291.958,-76.184,-178.000,10.371,149.541
C08115=1117.637,291.710,-76.154,-178.002,10.369,149.541
C08116=1117.640,291.462,-76.122,-178.005,10.367,149.541
C08117=1117.645,291.214,-76.091,-178.008,10.364,149.541
C08118=1117.648,290.966,-76.061,-178.012,10.362,149.542
C08119=1117.652,290.718,-76.029,-178.015,10.359,149.542
C08120=1117.656,290.470,-75.998,-178.018,10.356,149.542
C08121=1117.661,290.222,-75.967,-178.021,10.354,149.542
C08122=1117.665,289.974,-75.936,-178.024,10.351,149.542
C08123=1117.669,289.726,-75.905,-178.027,10.349,149.542
C08124=1117.674,289.478,-75.874,-178.030,10.346,149.542
C08125=1117.677,289.230,-75.843,-178.033,10.344,149.543
C08126=1117.682,288.982,-75.812,-178.036,10.341,149.543
C08127=1117.686,288.733,-75.781,-178.039,10.339,149.543
C08128=1117.690,288.485,-75.750,-178.042,10.336,149.543
C08129=1117.694,288.238,-75.720,-178.045,10.334,149.544
C08130=1117.698,287.990,-75.688,-178.048,10.331,149.544
C08131=1117.702,287.742,-75.657,-178.052,10.329,149.544
C08132=1117.706,287.493,-75.626,-178.054,10.326,149.544
C08133=1117.710,287.245,-75.596,-178.057,10.323,149.544
C08134=1117.715,286.998,-75.565,-178.060,10.321,149.544
C08135=1117.719,286.749,-75.534,-178.063,10.319,149.544
C08136=1117.723,286.502,-75.502,-178.066,10.316,149.545
C08137=1117.727,286.253,-75.472,-178.069,10.313,149.545
C08138=1117.731,286.005,-75.441,-178.073,10.311,149.545
C08139=1117.736,285.757,-75.410,-178.076,10.308,149.545
C08140=1117.739,285.509,-75.380,-178.079,10.305,149.545
C08141=1117.744,285.261,-75.349,-178.082,10.303,149.546
C08142=1117.748,285.013,-75.318,-178.085,10.300,149.546
C08143=1117.752,284.765,-75.288,-178.088,10.299,149.546
C08144=1117.756,284.517,-75.257,-178.090,10.296,149.546
C08145=1117.761,284.269,-75.226,-178.094,10.293,149.546
C08146=1117.764,284.020,-75.196,-178.097,10.291,149.546
C08147=1117.769,283.772,-75.165,-178.100,10.288,149.547
C08148=1117.773,283.524,-75.134,-178.103,10.286,149.547
C08149=1117.777,283.277,-75.104,-178.106,10.283,149.547
C08150=1117.781,283.028,-75.073,-178.109,10.280,149.547
C08151=1117.785,282.781,-75.043,-178.112,10.278,149.547
C08152=1117.790,282.532,-75.013,-178.115,10.276,149.547
C08153=1117.794,282.283,-74.982,-178.118,10.273,149.548
C08154=1117.798,282.036,-74.951,-178.121,10.270,149.548
C08155=1117.802,281.788,-74.921,-178.124,10.268,149.548
C08156=1117.806,281.540,-74.890,-178.127,10.265,149.548
C08157=1117.810,281.327,-74.864,-178.130,10.263,149.548
C08158=1117.814,281.114,-74.838,-178.133,10.261,149.549
C08159=1117.818,280.901,-74.812,-178.136,10.258,149.549
C08160=1117.821,280.688,-74.786,-178.138,10.256,149.549
C08161=1117.824,280.475,-74.760,-178.141,10.254,149.549
C08162=1117.828,280.262,-74.733,-178.144,10.252,149.549
C08163=1117.831,280.050,-74.707,-178.147,10.249,149.549
C08164=1117.835,279.837,-74.682,-178.149,10.247,149.550
C08165=1117.839,279.588,-74.651,-178.152,10.245,149.550
C08166=1117.843,279.341,-74.621,-178.155,10.242,149.550
C08167=1117.847,279.092,-74.590,-178.159,10.239,149.550
C08168=1117.852,278.844,-74.561,-178.162,10.236,149.550
C08169=1117.856,278.596,-74.530,-178.165,10.233,149.550
C08170=1117.860,278.348,-74.500,-178.168,10.231,149.550
C08171=1117.865,278.099,-74.470,-178.171,10.228,149.551
C08172=1117.868,277.851,-74.439,-178.175,10.225,149.551
C08173=1117.872,277.603,-74.410,-178.178,10.223,149.551
C08174=1117.877,277.355,-74.379,-178.181,10.220,149.551
C08175=1117.881,277.107,-74.349,-178.184,10.218,149.551
C08176=1117.885,276.859,-74.319,-178.187,10.215,149.551
C08177=1117.890,276.611,-74.289,-178.190,10.212,149.552
C08178=1117.893,276.362,-74.259,-178.193,10.209,149.552
C08179=1117.897,276.114,-74.229,-178.196,10.207,149.552
C08180=1117.902,275.866,-74.199,-178.199,10.204,149.552
C08181=1117.906,275.618,-74.168,-178.202,10.201,149.552
C08182=1117.910,275.370,-74.139,-178.205,10.199,149.552
C08183=1117.915,275.122,-74.108,-178.208,10.196,149.552
C08184=1117.919,274.874,-74.079,-178.211,10.193,149.553
C08185=1117.923,274.626,-74.049,-178.214,10.191,149.553
C08186=1117.927,274.377,-74.018,-178.217,10.188,149.553
C08187=1117.931,274.129,-73.988,-178.220,10.185,149.553
C08188=1117.935,273.881,-73.959,-178.223,10.182,149.553
C08189=1117.939,273.633,-73.929,-178.226,10.180,149.553
C08190=1117.944,273.385,-73.898,-178.229,10.178,149.553
C08191=1117.948,273.136,-73.869,-178.231,10.175,149.553
C08192=1117.952,272.888,-73.839,-178.234,10.172,149.554
C08193=1117.956,272.640,-73.809,-178.237,10.170,149.554
C08194=1117.960,272.392,-73.780,-178.240,10.167,149.554
C08195=1117.965,272.144,-73.750,-178.243,10.164,149.554
C08196=1117.969,271.896,-73.720,-178.246,10.161,149.554
C08197=1117.973,271.648,-73.690,-178.249,10.159,149.554
C08198=1117.978,271.399,-73.661,-178.251,10.157,149.554
C08199=1117.982,271.151,-73.631,-178.254,10.154,149.554
C08200=1117.986,270.903,-73.600,-178.257,10.151,149.554
C08201=1117.991,270.655,-73.571,-178.260,10.148,149.555
C08202=1117.995,270.407,-73.542,-178.263,10.146,149.555
C08203=1117.999,270.158,-73.512,-178.265,10.144,149.555
C08204=1118.003,269.910,-73.483,-178.268,10.141,149.555
C08205=1118.007,269.662,-73.452,-178.271,10.138,149.555
C08206=1118.011,269.414,-73.423,-178.274,10.135,149.555
C08207=1118.015,269.166,-73.394,-178.277,10.133,149.555
C08208=1118.020,268.917,-73.363,-178.280,10.131,149.555
C08209=1118.024,268.669,-73.334,-178.282,10.128,149.555
C08210=1118.029,268.421,-73.305,-178.285,10.125,149.555
C08211=1118.033,268.172,-73.275,-178.288,10.123,149.556
C08212=1118.037,267.924,-73.246,-178.291,10.120,149.556
C08213=1118.040,267.711,-73.220,-178.293,10.118,149.556
C08214=1118.044,267.498,-73.195,-178.295,10.116,149.556
C08215=1118.047,267.285,-73.169,-178.298,10.114,149.556
C08216=1118.051,267.072,-73.144,-178.300,10.112,149.556
C08217=1118.055,266.859,-73.119,-178.303,10.110,149.556
C08218=1118.058,266.646,-73.094,-178.305,10.107,149.556
C08219=1118.062,266.433,-73.069,-178.307,10.105,149.556
C08220=1118.066,266.220,-73.043,-178.309,10.103,149.556
C08221=1118.070,265.972,-73.013,-178.312,10.101,149.557
C08222=1118.074,265.724,-72.984,-178.315,10.099,149.557
C08223=1118.078,265.475,-72.954,-178.317,10.096,149.557
C08224=1118.083,265.226,-72.926,-178.320,10.094,149.557
C08225=1118.087,264.978,-72.896,-178.323,10.091,149.557
C08226=1118.091,264.730,-72.867,-178.326,10.088,149.557
C08227=1118.096,264.482,-72.838,-178.328,10.086,149.557
C08228=1118.100,264.234,-72.808,-178.332,10.083,149.558
C08229=1118.104,263.986,-72.779,-178.335,10.080,149.558
C08230=1118.108,263.738,-72.749,-178.338,10.078,149.558
C08231=1118.112,263.490,-72.721,-178.342,10.074,149.558
C08232=1118.116,263.241,-72.692,-178.345,10.072,149.558
C08233=1118.121,262.992,-72.662,-178.348,10.069,149.558
C08234=1118.125,262.744,-72.633,-178.351,10.067,149.559
C08235=1118.130,262.497,-72.604,-178.355,10.063,149.559
C08236=1118.134,262.248,-72.574,-178.358,10.061,149.559
C08237=1118.138,261.999,-72.546,-178.361,10.058,149.559
C08238=1118.142,261.751,-72.516,-178.364,10.055,149.559
C08239=1118.146,261.503,-72.487,-178.367,10.052,149.559
C08240=1118.151,261.256,-72.458,-178.370,10.049,149.559
C08241=1118.155,261.007,-72.429,-178.374,10.046,149.560
C08242=1118.159,260.759,-72.400,-178.377,10.044,149.560
C08243=1118.163,260.510,-72.371,-178.380,10.041,149.560
C08244=1118.167,260.262,-72.342,-178.383,10.037,149.560
C08245=1118.171,260.013,-72.313,-178.386,10.035,149.560
C08246=1118.176,259.765,-72.285,-178.389,10.032,149.560
C08247=1118.181,259.517,-72.255,-178.392,10.029,149.560
C08248=1118.184,259.269,-72.226,-178.395,10.026,149.560
C08249=1118.189,259.020,-72.198,-178.398,10.024,149.560
C08250=1118.193,258.773,-72.168,-178.401,10.021,149.561
C08251=1118.198,258.524,-72.140,-178.404,10.018,149.561
C08252=1118.201,258.276,-72.111,-178.406,10.015,149.561
C08253=1118.206,258.027,-72.082,-178.409,10.012,149.561
C08254=1118.211,257.779,-72.053,-178.412,10.009,149.561
C08255=1118.214,257.531,-72.025,-178.415,10.007,149.561
C08256=1118.219,257.282,-71.995,-178.418,10.004,149.561
C08257=1118.223,257.034,-71.967,-178.421,10.001,149.561
C08258=1118.227,256.786,-71.938,-178.424,9.998,149.561
C08259=1118.232,256.537,-71.909,-178.426,9.995,149.561
C08260=1118.236,256.289,-71.880,-178.429,9.993,149.561
C08261=1118.240,256.041,-71.852,-178.432,9.990,149.561
C08262=1118.245,255.792,-71.823,-178.433,9.988,149.561
C08263=1118.249,255.544,-71.794,-178.434,9.986,149.561
C08264=1118.253,255.296,-71.766,-178.435,9.984,149.561
C08265=1118.257,255.048,-71.737,-178.437,9.983,149.561
C08266=1118.261,254.799,-71.709,-178.438,9.981,149.561
C08267=1118.266,254.550,-71.680,-178.440,9.979,149.561
C08268=1118.270,254.303,-71.651,-178.442,9.977,149.561
C08269=1118.273,254.089,-71.627,-178.443,9.975,149.561
C08270=1118.278,253.876,-71.602,-178.445,9.974,149.561
C08271=1118.281,253.663,-71.577,-178.447,9.972,149.561
C08272=1118.285,253.450,-71.553,-178.448,9.970,149.561
C08273=1118.288,253.237,-71.528,-178.450,9.968,149.561
C08274=1118.292,253.024,-71.504,-178.453,9.966,149.561
C08275=1118.296,252.810,-71.480,-178.454,9.965,149.561
C08276=1118.300,252.597,-71.455,-178.456,9.963,149.561
C08277=1118.304,252.349,-71.427,-178.460,9.960,149.562
C08278=1118.308,252.101,-71.397,-178.463,9.958,149.562
C08279=1118.312,251.853,-71.369,-178.466,9.955,149.562
C08280=1118.317,251.604,-71.341,-178.469,9.953,149.562
C08281=1118.320,251.355,-71.313,-178.472,9.950,149.562
C08282=1118.326,251.107,-71.284,-178.475,9.947,149.562
C08283=1118.329,250.859,-71.255,-178.478,9.945,149.563
C08284=1118.334,250.611,-71.227,-178.482,9.942,149.563
C08285=1118.338,250.362,-71.199,-178.486,9.938,149.563
C08286=1118.342,250.113,-71.170,-178.490,9.935,149.563
C08287=1118.347,249.866,-71.142,-178.494,9.932,149.564
C08288=1118.351,249.617,-71.114,-178.498,9.929,149.564
C08289=1118.355,249.369,-71.086,-178.502,9.926,149.564
C08290=1118.359,249.121,-71.057,-178.507,9.922,149.565
C08291=1118.363,248.872,-71.028,-178.511,9.919,149.565
C08292=1118.368,248.624,-71.000,-178.515,9.915,149.565
C08293=1118.372,248.375,-70.972,-178.520,9.911,149.565
C08294=1118.377,248.127,-70.944,-178.525,9.907,149.566
C08295=1118.380,247.879,-70.916,-178.529,9.903,149.566
C08296=1118.386,247.630,-70.888,-178.535,9.898,149.566
C08297=1118.390,247.381,-70.860,-178.538,9.894,149.566
C08298=1118.394,247.134,-70.832,-178.540,9.892,149.566
C08299=1118.398,246.885,-70.803,-178.542,9.890,149.566
C08300=1118.403,246.637,-70.776,-178.543,9.887,149.566
C08301=1118.406,246.388,-70.747,-178.545,9.885,149.566
C08302=1118.411,246.140,-70.720,-178.547,9.882,149.566
C08303=1118.415,245.891,-70.691,-178.550,9.879,149.566
C08304=1118.420,245.644,-70.663,-178.552,9.877,149.566
C08305=1118.424,245.394,-70.636,-178.553,9.875,149.566
C08306=1118.429,245.146,-70.607,-178.555,9.872,149.566
C08307=1118.433,244.898,-70.579,-178.557,9.870,149.566
C08308=1118.437,244.650,-70.551,-178.559,9.868,149.565
C08309=1118.441,244.402,-70.524,-178.562,9.865,149.565
C08310=1118.446,244.152,-70.496,-178.564,9.863,149.566
C08311=1118.450,243.904,-70.468,-178.566,9.860,149.565
C08312=1118.454,243.656,-70.440,-178.568,9.858,149.565
C08313=1118.458,243.408,-70.412,-178.570,9.855,149.565
C08314=1118.463,243.159,-70.385,-178.573,9.853,149.565
C08315=1118.468,242.911,-70.356,-178.574,9.850,149.565
C08316=1118.471,242.662,-70.328,-178.577,9.847,149.565
C08317=1118.476,242.414,-70.300,-178.579,9.845,149.565
C08318=1118.480,242.166,-70.273,-178.581,9.843,149.565
C08319=1118.484,241.917,-70.245,-178.584,9.840,149.566
C08320=1118.488,241.669,-70.217,-178.586,9.838,149.565
C08321=1118.493,241.420,-70.189,-178.588,9.836,149.565
C08322=1118.498,241.172,-70.161,-178.591,9.833,149.566
C08323=1118.502,240.924,-70.134,-178.593,9.831,149.566
C08324=1118.506,240.675,-70.106,-178.596,9.828,149.566
C08325=1118.510,240.462,-70.083,-178.598,9.826,149.566
C08326=1118.513,240.249,-70.059,-178.600,9.824,149.566
C08327=1118.517,240.035,-70.035,-178.602,9.822,149.566
C08328=1118.521,239.822,-70.011,-178.604,9.819,149.566
C08329=1118.525,239.609,-69.988,-178.606,9.817,149.566
C08330=1118.528,239.395,-69.964,-178.608,9.815,149.566
C08331=1118.532,239.182,-69.940,-178.611,9.813,149.566
C08332=1118.536,238.969,-69.916,-178.613,9.811,149.566
C08333=1118.540,238.720,-69.888,-178.616,9.808,149.566
C08334=1118.545,238.471,-69.861,-178.618,9.806,149.566
C08335=1118.549,238.224,-69.833,-178.621,9.803,149.566
C08336=1118.553,237.974,-69.806,-178.623,9.801,149.566
C08337=1118.557,237.727,-69.778,-178.626,9.798,149.566
C08338=1118.562,237.478,-69.751,-178.629,9.795,149.566
C08339=1118.566,237.229,-69.723,-178.631,9.793,149.567
C08340=1118.570,236.981,-69.696,-178.634,9.791,149.567
C08341=1118.575,236.733,-69.668,-178.636,9.787,149.567
C08342=1118.579,236.485,-69.641,-178.639,9.785,149.567
C08343=1118.583,236.235,-69.614,-178.642,9.782,149.567
C08344=1118.588,235.988,-69.586,-178.645,9.780,149.567
C08345=1118.592,235.739,-69.559,-178.648,9.777,149.567
C08346=1118.596,235.490,-69.531,-178.650,9.775,149.567
C08347=1118.601,235.242,-69.504,-178.653,9.772,149.567
C08348=1118.606,234.993,-69.476,-178.656,9.769,149.567
C08349=1118.610,234.746,-69.449,-178.659,9.766,149.567
C08350=1118.614,234.496,-69.421,-178.662,9.763,149.568
C08351=1118.619,234.248,-69.394,-178.665,9.760,149.568
C08352=1118.623,233.999,-69.367,-178.668,9.758,149.568
C08353=1118.627,233.752,-69.340,-178.671,9.755,149.568
C08354=1118.631,233.503,-69.313,-178.674,9.752,149.568
C08355=1118.636,233.254,-69.285,-178.677,9.749,149.568
C08356=1118.640,233.006,-69.258,-178.679,9.747,149.568
C08357=1118.645,232.758,-69.231,-178.682,9.744,149.568
C08358=1118.649,232.509,-69.203,-178.685,9.741,149.568
C08359=1118.653,232.260,-69.176,-178.688,9.738,149.569
C08360=1118.657,232.012,-69.150,-178.691,9.735,149.569
C08361=1118.662,231.763,-69.123,-178.694,9.732,149.569
C08362=1118.666,231.516,-69.095,-178.697,9.729,149.569
C08363=1118.670,231.266,-69.067,-178.700,9.726,149.569
C08364=1118.675,231.018,-69.040,-178.704,9.723,149.569
C08365=1118.680,230.769,-69.013,-178.707,9.720,149.569
C08366=1118.683,230.521,-68.987,-178.710,9.717,149.569
C08367=1118.688,230.273,-68.960,-178.713,9.713,149.569
C08368=1118.693,230.024,-68.933,-178.716,9.711,149.569
C08369=1118.697,229.775,-68.905,-178.719,9.707,149.570
C08370=1118.701,229.527,-68.879,-178.722,9.704,149.570
C08371=1118.705,229.278,-68.852,-178.725,9.702,149.570
C08372=1118.710,229.030,-68.825,-178.729,9.698,149.570
C08373=1118.714,228.782,-68.798,-178.731,9.695,149.570
C08374=1118.719,228.533,-68.771,-178.735,9.691,149.570
C08375=1118.723,228.285,-68.744,-178.738,9.689,149.570
C08376=1118.727,228.035,-68.717,-178.741,9.686,149.570
C08377=1118.731,227.787,-68.690,-178.744,9.682,149.570
C08378=1118.736,227.539,-68.663,-178.747,9.679,149.570
C08379=1118.741,227.290,-68.636,-178.750,9.675,149.570
C08380=1118.745,227.042,-68.610,-178.753,9.672,149.570
C08381=1118.749,226.828,-68.587,-178.756,9.670,149.570
C08382=1118.753,226.615,-68.564,-178.758,9.667,149.570
C08383=1118.756,226.402,-68.541,-178.761,9.665,149.570
C08384=1118.760,226.188,-68.518,-178.763,9.661,149.570
C08385=1118.764,225.975,-68.496,-178.765,9.659,149.570
C08386=1118.767,225.762,-68.472,-178.768,9.656,149.570
C08387=1118.771,225.548,-68.449,-178.770,9.653,149.570
C08388=1118.776,225.334,-68.426,-178.772,9.651,149.570
C08389=1118.779,225.086,-68.400,-178.776,9.647,149.570
C08390=1118.783,224.837,-68.373,-178.778,9.644,149.570
C08391=1118.788,224.588,-68.347,-178.781,9.641,149.570
C08392=1118.792,224.340,-68.320,-178.784,9.638,149.570
C08393=1118.796,224.092,-68.293,-178.786,9.635,149.570
C08394=1118.801,223.843,-68.266,-178.789,9.631,149.570
C08395=1118.806,223.594,-68.240,-178.792,9.628,149.570
C08396=1118.810,223.346,-68.213,-178.795,9.625,149.570
C08397=1118.814,223.097,-68.186,-178.797,9.622,149.570
C08398=1118.819,222.848,-68.161,-178.800,9.619,149.570
C08399=1118.823,222.600,-68.134,-178.802,9.616,149.570
C08400=1118.828,222.351,-68.108,-178.805,9.613,149.570
C08401=1118.832,222.104,-68.082,-178.807,9.610,149.570
C08402=1118.837,221.855,-68.055,-178.810,9.607,149.570
C08403=1118.841,221.606,-68.029,-178.812,9.603,149.570
C08404=1118.846,221.358,-68.002,-178.815,9.600,149.570
C08405=1118.850,221.109,-67.976,-178.817,9.597,149.569
C08406=1118.855,220.861,-67.949,-178.820,9.594,149.569
C08407=1118.859,220.612,-67.923,-178.822,9.591,149.569
C08408=1118.863,220.364,-67.897,-178.825,9.588,149.569
C08409=1118.868,220.114,-67.870,-178.827,9.584,149.569
C08410=1118.872,219.866,-67.844,-178.830,9.581,149.569
C08411=1118.877,219.617,-67.818,-178.832,9.578,149.569
C08412=1118.880,219.369,-67.791,-178.835,9.575,149.569
C08413=1118.885,219.120,-67.765,-178.837,9.572,149.569
C08414=1118.889,218.872,-67.738,-178.840,9.569,149.569
C08415=1118.894,218.623,-67.713,-178.841,9.566,149.568
C08416=1118.898,218.375,-67.687,-178.844,9.563,149.568
C08417=1118.903,218.126,-67.660,-178.846,9.560,149.568
C08418=1118.907,217.877,-67.634,-178.849,9.557,149.568
C08419=1118.911,217.629,-67.608,-178.851,9.553,149.568
C08420=1118.916,217.380,-67.582,-178.853,9.551,149.568
C08421=1118.920,217.131,-67.556,-178.855,9.548,149.568
C08422=1118.924,216.883,-67.529,-178.858,9.545,149.568
C08423=1118.928,216.634,-67.504,-178.859,9.542,149.568
C08424=1118.934,216.386,-67.478,-178.862,9.539,149.567
C08425=1118.938,216.138,-67.451,-178.864,9.536,149.567
C08426=1118.942,215.889,-67.425,-178.866,9.533,149.567
C08427=1118.946,215.640,-67.400,-178.868,9.530,149.567
C08428=1118.951,215.391,-67.373,-178.870,9.528,149.567
C08429=1118.955,215.143,-67.347,-178.872,9.524,149.567
C08430=1118.960,214.894,-67.321,-178.875,9.521,149.567
C08431=1118.964,214.646,-67.296,-178.877,9.519,149.567
C08432=1118.969,214.397,-67.269,-178.879,9.515,149.566
C08433=1118.973,214.149,-67.243,-178.881,9.513,149.566
C08434=1118.977,213.900,-67.217,-178.883,9.511,149.566
C08435=1118.982,213.651,-67.191,-178.885,9.507,149.566
C08436=1118.987,213.403,-67.166,-178.887,9.505,149.566
C08437=1118.991,213.189,-67.143,-178.889,9.502,149.566
C08438=1118.994,212.976,-67.121,-178.891,9.499,149.566
C08439=1118.998,212.762,-67.099,-178.893,9.497,149.566
C08440=1119.001,212.548,-67.077,-178.895,9.495,149.566
C08441=1119.006,212.335,-67.054,-178.897,9.492,149.566
C08442=1119.009,212.121,-67.033,-178.899,9.489,149.566
C08443=1119.013,211.908,-67.011,-178.901,9.487,149.566
C08444=1119.017,211.694,-66.988,-178.903,9.485,149.566
C08445=1119.021,211.446,-66.962,-178.906,9.482,149.566
C08446=1119.026,211.197,-66.936,-178.909,9.479,149.566
C08447=1119.030,210.948,-66.911,-178.910,9.476,149.566
C08448=1119.035,210.700,-66.885,-178.913,9.473,149.566
C08449=1119.039,210.451,-66.860,-178.915,9.470,149.566
C08450=1119.044,210.202,-66.833,-178.918,9.468,149.566
C08451=1119.049,209.954,-66.808,-178.921,9.464,149.566
C08452=1119.053,209.705,-66.782,-178.923,9.461,149.566
C08453=1119.057,209.456,-66.756,-178.926,9.459,149.566
C08454=1119.061,209.208,-66.731,-178.928,9.456,149.566
C08455=1119.066,208.959,-66.705,-178.931,9.453,149.566
C08456=1119.070,208.711,-66.679,-178.934,9.450,149.566
C08457=1119.075,208.462,-66.654,-178.937,9.448,149.566
C08458=1119.079,208.214,-66.628,-178.939,9.445,149.566
C08459=1119.084,207.965,-66.603,-178.942,9.442,149.566
C08460=1119.088,207.715,-66.577,-178.945,9.439,149.566
C08461=1119.093,207.467,-66.552,-178.948,9.436,149.566
C08462=1119.097,207.219,-66.526,-178.950,9.434,149.566
C08463=1119.101,206.970,-66.501,-178.953,9.431,149.566
C08464=1119.106,206.722,-66.475,-178.955,9.428,149.566
C08465=1119.110,206.473,-66.449,-178.958,9.425,149.566
C08466=1119.115,206.223,-66.424,-178.961,9.422,149.566
C08467=1119.120,205.975,-66.399,-178.964,9.420,149.567
C08468=1119.124,205.727,-66.373,-178.967,9.417,149.567
C08469=1119.128,205.478,-66.348,-178.969,9.414,149.567
C08470=1119.132,205.230,-66.323,-178.972,9.411,149.567
C08471=1119.137,204.981,-66.298,-178.975,9.408,149.567
C08472=1119.142,204.732,-66.272,-178.979,9.405,149.567
C08473=1119.146,204.484,-66.247,-178.981,9.402,149.567
C08474=1119.150,204.234,-66.222,-178.984,9.399,149.567
C08475=1119.155,203.986,-66.196,-178.987,9.396,149.567
C08476=1119.160,203.737,-66.170,-178.990,9.393,149.567
C08477=1119.165,203.489,-66.146,-178.993,9.390,149.567
C08478=1119.168,203.240,-66.121,-178.996,9.387,149.568
C08479=1119.172,202.991,-66.095,-178.999,9.385,149.568
C08480=1119.177,202.743,-66.070,-179.002,9.381,149.568
C08481=1119.182,202.494,-66.044,-179.005,9.378,149.568
C08482=1119.187,202.245,-66.020,-179.008,9.375,149.568
C08483=1119.190,201.997,-65.995,-179.011,9.373,149.568
C08484=1119.195,201.748,-65.969,-179.014,9.369,149.568
C08485=1119.200,201.499,-65.944,-179.017,9.366,149.568
C08486=1119.205,201.251,-65.919,-179.020,9.363,149.568
C08487=1119.208,201.002,-65.894,-179.023,9.360,149.568
C08488=1119.213,200.754,-65.869,-179.026,9.357,149.569
C08489=1119.218,200.504,-65.844,-179.029,9.354,149.569
C08490=1119.222,200.256,-65.819,-179.032,9.350,149.569
C08491=1119.226,200.007,-65.794,-179.035,9.348,149.569
C08492=1119.231,199.758,-65.769,-179.039,9.344,149.569
C08493=1119.236,199.473,-65.740,-179.042,9.341,149.569
C08494=1119.242,199.188,-65.712,-179.046,9.337,149.569
C08495=1119.246,198.903,-65.684,-179.049,9.333,149.569
C08496=1119.251,198.618,-65.655,-179.053,9.330,149.569
C08497=1119.256,198.369,-65.630,-179.056,9.326,149.569
C08498=1119.261,198.121,-65.605,-179.059,9.323,149.569
C08499=1119.265,197.872,-65.580,-179.063,9.320,149.570
C08500=1119.270,197.624,-65.555,-179.065,9.317,149.570
C08501=1119.274,197.374,-65.531,-179.069,9.313,149.570
C08502=1119.279,197.126,-65.506,-179.072,9.309,149.570
C08503=1119.282,196.877,-65.481,-179.075,9.306,149.570
C08504=1119.287,196.628,-65.456,-179.078,9.303,149.570
C08505=1119.293,196.380,-65.431,-179.081,9.299,149.570
C08506=1119.296,196.131,-65.407,-179.083,9.297,149.570
C08507=1119.301,195.882,-65.382,-179.085,9.293,149.569
C08508=1119.305,195.633,-65.357,-179.087,9.291,149.569
C08509=1119.310,195.385,-65.332,-179.089,9.288,149.569
C08510=1119.314,195.136,-65.308,-179.091,9.286,149.569
C08511=1119.319,194.887,-65.283,-179.093,9.283,149.569
C08512=1119.323,194.638,-65.259,-179.095,9.280,149.569
C08513=1119.328,194.389,-65.234,-179.097,9.278,149.569
C08514=1119.332,194.141,-65.209,-179.098,9.275,149.569
C08515=1119.337,193.892,-65.185,-179.101,9.272,149.569
C08516=1119.341,193.643,-65.160,-179.102,9.269,149.568
C08517=1119.346,193.395,-65.136,-179.104,9.267,149.568
C08518=1119.350,193.146,-65.112,-179.106,9.264,149.568
C08519=1119.355,192.897,-65.087,-179.108,9.261,149.568
C08520=1119.359,192.648,-65.063,-179.110,9.259,149.568
C08521=1119.365,192.400,-65.038,-179.112,9.255,149.568
C08522=1119.368,192.151,-65.013,-179.114,9.253,149.568
C08523=1119.373,191.902,-64.989,-179.116,9.251,149.568
C08524=1119.378,191.653,-64.965,-179.119,9.248,149.568
C08525=1119.382,191.404,-64.940,-179.121,9.245,149.568
C08526=1119.387,191.156,-64.916,-179.123,9.242,149.568
C08527=1119.391,190.907,-64.891,-179.125,9.240,149.567
C08528=1119.396,190.658,-64.866,-179.127,9.236,149.567
C08529=1119.400,190.409,-64.842,-179.129,9.234,149.567
C08530=1119.405,190.161,-64.818,-179.132,9.231,149.567
C08531=1119.410,189.912,-64.794,-179.133,9.229,149.567
C08532=1119.413,189.663,-64.769,-179.136,9.226,149.567
C08533=1119.419,189.414,-64.745,-179.138,9.223,149.567
C08534=1119.423,189.166,-64.720,-179.140,9.220,149.567
C08535=1119.427,188.917,-64.696,-179.142,9.218,149.567
C08536=1119.432,188.668,-64.671,-179.145,9.215,149.567
C08537=1119.436,188.420,-64.647,-179.147,9.212,149.567
C08538=1119.441,188.171,-64.624,-179.149,9.209,149.567
C08539=1119.446,187.921,-64.599,-179.152,9.206,149.567
C08540=1119.450,187.673,-64.575,-179.154,9.204,149.567
C08541=1119.457,187.282,-64.537,-179.157,9.199,149.567
C08542=1119.464,186.890,-64.499,-179.161,9.194,149.567
C08543=1119.471,186.500,-64.461,-179.165,9.190,149.567
C08544=1119.479,186.108,-64.423,-179.169,9.185,149.567
C08545=1119.482,185.895,-64.402,-179.171,9.183,149.567
C08546=1119.486,185.681,-64.381,-179.173,9.181,149.567
C08547=1119.491,185.467,-64.360,-179.175,9.178,149.567
C08548=1119.494,185.253,-64.340,-179.177,9.175,149.567
C08549=1119.498,185.040,-64.319,-179.179,9.173,149.567
C08550=1119.502,184.825,-64.298,-179.181,9.171,149.567
C08551=1119.505,184.612,-64.278,-179.184,9.168,149.567
C08552=1119.510,184.398,-64.257,-179.186,9.165,149.567
C08553=1119.514,184.149,-64.233,-179.188,9.162,149.566
C08554=1119.518,183.900,-64.210,-179.191,9.159,149.566
C08555=1119.524,183.652,-64.185,-179.194,9.156,149.567
C08556=1119.528,183.403,-64.161,-179.196,9.153,149.567
C08557=1119.533,183.154,-64.137,-179.199,9.150,149.567
C08558=1119.537,182.906,-64.113,-179.201,9.147,149.566
C08559=1119.542,182.657,-64.090,-179.204,9.144,149.566
C08560=1119.545,182.408,-64.066,-179.206,9.141,149.566
C08561=1119.550,182.159,-64.042,-179.209,9.138,149.566
C08562=1119.555,181.910,-64.018,-179.211,9.135,149.566
C08563=1119.560,181.661,-63.994,-179.214,9.132,149.566
C08564=1119.564,181.412,-63.970,-179.217,9.129,149.566
C08565=1119.569,181.164,-63.946,-179.219,9.126,149.566
C08566=1119.574,180.915,-63.923,-179.222,9.123,149.566
C08567=1119.578,180.667,-63.899,-179.224,9.119,149.566
C08568=1119.582,180.417,-63.875,-179.227,9.116,149.566
C08569=1119.587,180.168,-63.852,-179.230,9.112,149.566
C08570=1119.591,179.919,-63.827,-179.232,9.109,149.566
C08571=1119.596,179.670,-63.804,-179.235,9.107,149.566
C08572=1119.600,179.422,-63.780,-179.239,9.103,149.566
C08573=1119.605,179.173,-63.757,-179.241,9.100,149.566
C08574=1119.609,178.924,-63.733,-179.243,9.097,149.566
C08575=1119.614,178.675,-63.709,-179.245,9.094,149.566
C08576=1119.619,178.426,-63.686,-179.247,9.091,149.566
C08577=1119.623,178.178,-63.662,-179.249,9.088,149.566
C08578=1119.628,177.929,-63.638,-179.252,9.085,149.566
C08579=1119.632,177.680,-63.615,-179.253,9.082,149.565
C08580=1119.637,177.431,-63.591,-179.256,9.079,149.565
C08581=1119.642,177.182,-63.568,-179.258,9.076,149.565
C08582=1119.646,176.933,-63.544,-179.260,9.073,149.565
C08583=1119.651,176.684,-63.521,-179.262,9.070,149.565
C08584=1119.655,176.436,-63.497,-179.264,9.068,149.565
C08585=1119.660,176.187,-63.474,-179.266,9.064,149.565
C08586=1119.665,175.938,-63.450,-179.269,9.061,149.565
C08587=1119.669,175.689,-63.427,-179.271,9.059,149.565
C08588=1119.673,175.441,-63.403,-179.273,9.056,149.565
C08589=1119.678,175.192,-63.380,-179.275,9.052,149.564
C08590=1119.683,174.943,-63.357,-179.277,9.050,149.564
C08591=1119.687,174.694,-63.333,-179.280,9.047,149.564
C08592=1119.692,174.445,-63.310,-179.282,9.043,149.564
C08593=1119.696,174.196,-63.286,-179.284,9.040,149.564
C08594=1119.701,173.947,-63.262,-179.286,9.038,149.564
C08595=1119.705,173.698,-63.240,-179.288,9.034,149.564
C08596=1119.710,173.449,-63.216,-179.291,9.031,149.564
C08597=1119.714,173.200,-63.193,-179.293,9.029,149.564
C08598=1119.719,172.951,-63.170,-179.295,9.026,149.563
C08599=1119.724,172.702,-63.146,-179.297,9.022,149.563
C08600=1119.728,172.453,-63.123,-179.299,9.020,149.563
C08601=1119.732,172.240,-63.103,-179.302,9.017,149.563
C08602=1119.736,172.026,-63.083,-179.303,9.014,149.563
C08603=1119.741,171.812,-63.063,-179.305,9.012,149.563
C08604=1119.744,171.598,-63.043,-179.307,9.010,149.563
C08605=1119.747,171.384,-63.023,-179.309,9.007,149.563
C08606=1119.752,171.171,-63.003,-179.311,9.004,149.563
C08607=1119.756,170.956,-62.983,-179.313,9.001,149.563
C08608=1119.760,170.743,-62.964,-179.315,8.999,149.563
C08609=1119.765,170.494,-62.940,-179.317,8.996,149.563
C08610=1119.769,170.245,-62.917,-179.319,8.993,149.562
C08611=1119.773,169.996,-62.894,-179.321,8.990,149.562
C08612=1119.778,169.747,-62.871,-179.324,8.987,149.562
C08613=1119.783,169.498,-62.847,-179.326,8.984,149.562
C08614=1119.787,169.249,-62.825,-179.328,8.981,149.562
C08615=1119.792,169.001,-62.802,-179.331,8.977,149.562
C08616=1119.797,168.752,-62.778,-179.332,8.975,149.562
C08617=1119.801,168.503,-62.755,-179.335,8.972,149.562
C08618=1119.805,168.254,-62.732,-179.337,8.968,149.562
C08619=1119.810,168.005,-62.710,-179.340,8.965,149.562
C08620=1119.815,167.755,-62.686,-179.342,8.962,149.561
C08621=1119.820,167.507,-62.664,-179.344,8.960,149.561
C08622=1119.824,167.258,-62.640,-179.346,8.956,149.561
C08623=1119.829,167.009,-62.617,-179.348,8.953,149.561
C08624=1119.833,166.761,-62.594,-179.351,8.950,149.561
C08625=1119.838,166.511,-62.572,-179.353,8.947,149.561
C08626=1119.842,166.263,-62.549,-179.355,8.944,149.561
C08627=1119.847,166.014,-62.526,-179.357,8.941,149.561
C08628=1119.852,165.765,-62.503,-179.360,8.938,149.561
C08629=1119.856,165.516,-62.481,-179.362,8.934,149.561
C08630=1119.861,165.267,-62.457,-179.365,8.931,149.561
C08631=1119.865,165.019,-62.435,-179.367,8.928,149.560
C08632=1119.870,164.770,-62.411,-179.369,8.925,149.560
C08633=1119.874,164.520,-62.389,-179.372,8.922,149.560
C08634=1119.879,164.271,-62.366,-179.374,8.919,149.560
C08635=1119.884,164.023,-62.343,-179.376,8.916,149.560
C08636=1119.889,163.773,-62.321,-179.378,8.913,149.560
C08637=1119.893,163.524,-62.298,-179.381,8.909,149.560
C08638=1119.897,163.276,-62.275,-179.383,8.906,149.560
C08639=1119.903,163.027,-62.253,-179.385,8.903,149.560
C08640=1119.907,162.778,-62.230,-179.387,8.899,149.559
C08641=1119.911,162.529,-62.208,-179.390,8.896,149.559
C08642=1119.916,162.280,-62.184,-179.392,8.893,149.559
C08643=1119.920,162.032,-62.162,-179.395,8.890,149.559
C08644=1119.925,161.782,-62.139,-179.397,8.887,149.559
C08645=1119.929,161.533,-62.117,-179.400,8.883,149.559
C08646=1119.935,161.284,-62.094,-179.402,8.880,149.559
C08647=1119.939,161.036,-62.072,-179.404,8.877,149.559
C08648=1119.944,160.786,-62.049,-179.406,8.874,149.558
C08649=1119.948,160.538,-62.026,-179.408,8.871,149.558
C08650=1119.953,160.289,-62.004,-179.410,8.868,149.558
C08651=1119.957,160.040,-61.981,-179.413,8.864,149.558
C08652=1119.962,159.791,-61.959,-179.415,8.861,149.558
C08653=1119.967,159.542,-61.936,-179.417,8.858,149.558
C08654=1119.971,159.293,-61.914,-179.420,8.855,149.558
C08655=1119.976,159.044,-61.892,-179.422,8.851,149.558
C08656=1119.981,158.795,-61.869,-179.425,8.847,149.558
C08657=1119.985,158.581,-61.850,-179.427,8.845,149.557
C08658=1119.989,158.367,-61.831,-179.428,8.842,149.557
C08659=1119.993,158.153,-61.811,-179.431,8.839,149.557
C08660=1119.996,157.939,-61.792,-179.432,8.837,149.557
C08661=1120.000,157.725,-61.773,-179.435,8.833,149.557
C08662=1120.004,157.511,-61.754,-179.436,8.831,149.557
C08663=1120.008,157.297,-61.735,-179.439,8.828,149.557
C08664=1120.012,157.083,-61.715,-179.440,8.825,149.557
C08665=1120.016,156.834,-61.693,-179.444,8.821,149.557
C08666=1120.022,156.585,-61.671,-179.446,8.818,149.556
C08667=1120.026,156.336,-61.648,-179.448,8.814,149.556
C08668=1120.031,156.087,-61.627,-179.450,8.811,149.556
C08669=1120.036,155.838,-61.604,-179.453,8.808,149.556
C08670=1120.041,155.589,-61.582,-179.455,8.804,149.556
C08671=1120.045,155.340,-61.560,-179.457,8.801,149.556
C08672=1120.049,155.091,-61.538,-179.459,8.798,149.556
C08673=1120.055,154.842,-61.515,-179.462,8.795,149.555
C08674=1120.059,154.593,-61.493,-179.465,8.790,149.555
C08675=1120.064,154.344,-61.471,-179.467,8.787,149.555
C08676=1120.068,154.095,-61.449,-179.469,8.784,149.555
C08677=1120.073,153.847,-61.427,-179.471,8.780,149.555
C08678=1120.078,153.597,-61.404,-179.474,8.777,149.555
C08679=1120.082,153.348,-61.383,-179.476,8.774,149.554
C08680=1120.087,153.099,-61.361,-179.479,8.769,149.554
C08681=1120.092,152.850,-61.339,-179.481,8.766,149.554
C08682=1120.096,152.601,-61.317,-179.483,8.763,149.554
C08683=1120.101,152.352,-61.295,-179.485,8.759,149.554
C08684=1120.105,152.103,-61.273,-179.488,8.755,149.554
C08685=1120.111,151.854,-61.251,-179.491,8.752,149.553
C08686=1120.115,151.605,-61.229,-179.493,8.748,149.553
C08687=1120.120,151.356,-61.207,-179.495,8.745,149.553
C08688=1120.124,151.107,-61.185,-179.498,8.741,149.553
C08689=1120.129,150.858,-61.163,-179.500,8.738,149.553
C08690=1120.133,150.609,-61.141,-179.502,8.734,149.552
C08691=1120.138,150.360,-61.120,-179.505,8.731,149.552
C08692=1120.143,150.112,-61.098,-179.507,8.727,149.552
C08693=1120.147,149.862,-61.076,-179.509,8.723,149.552
C08694=1120.152,149.614,-61.054,-179.511,8.720,149.552
C08695=1120.156,149.364,-61.032,-179.514,8.716,149.552
C08696=1120.161,149.116,-61.011,-179.517,8.712,149.551
C08697=1120.165,148.866,-60.989,-179.519,8.709,149.551
C08698=1120.170,148.618,-60.967,-179.521,8.705,149.551
C08699=1120.175,148.369,-60.945,-179.524,8.701,149.551
C08700=1120.180,148.119,-60.924,-179.526,8.698,149.551
C08701=1120.185,147.870,-60.902,-179.528,8.693,149.550
C08702=1120.189,147.621,-60.880,-179.531,8.690,149.550
C08703=1120.194,147.372,-60.858,-179.533,8.687,149.550
C08704=1120.199,147.124,-60.837,-179.536,8.683,149.550
C08705=1120.203,146.874,-60.815,-179.538,8.679,149.550
C08706=1120.208,146.625,-60.794,-179.540,8.675,149.549
C08707=1120.213,146.376,-60.772,-179.543,8.671,149.549
C08708=1120.217,146.127,-60.750,-179.545,8.668,149.549
C08709=1120.222,145.878,-60.729,-179.547,8.664,149.549
C08710=1120.227,145.629,-60.707,-179.549,8.660,149.548
C08711=1120.231,145.380,-60.685,-179.552,8.656,149.548
C08712=1120.237,145.131,-60.664,-179.554,8.652,149.548
C08713=1120.240,144.917,-60.646,-179.556,8.650,149.548
C08714=1120.244,144.703,-60.627,-179.557,8.647,149.547
C08715=1120.248,144.489,-60.609,-179.558,8.644,149.547
C08716=1120.252,144.275,-60.590,-179.560,8.640,149.547
C08717=1120.256,144.060,-60.572,-179.561,8.637,149.546
C08718=1120.260,143.846,-60.553,-179.563,8.635,149.546
C08719=1120.264,143.633,-60.535,-179.564,8.631,149.546
C08720=1120.268,143.418,-60.517,-179.565,8.629,149.545
C08721=1120.273,143.169,-60.495,-179.567,8.626,149.545
C08722=1120.277,142.920,-60.474,-179.568,8.622,149.545
C08723=1120.282,142.671,-60.453,-179.570,8.618,149.544
C08724=1120.287,142.422,-60.431,-179.571,8.616,149.544
C08725=1120.292,142.172,-60.410,-179.573,8.612,149.544
C08726=1120.296,141.924,-60.388,-179.574,8.609,149.544
C08727=1120.301,141.675,-60.368,-179.576,8.605,149.543
C08728=1120.306,141.426,-60.346,-179.577,8.602,149.543
C08729=1120.310,141.176,-60.325,-179.579,8.599,149.542
C08730=1120.315,140.928,-60.303,-179.581,8.595,149.542
C08731=1120.320,140.679,-60.283,-179.582,8.592,149.542
C08732=1120.324,140.430,-60.261,-179.584,8.588,149.542
C08733=1120.329,140.180,-60.240,-179.585,8.585,149.541
C08734=1120.334,139.931,-60.218,-179.587,8.582,149.541
C08735=1120.338,139.682,-60.198,-179.589,8.579,149.541
C08736=1120.343,139.433,-60.177,-179.590,8.575,149.540
C08737=1120.348,139.184,-60.155,-179.592,8.572,149.540
C08738=1120.352,138.935,-60.134,-179.593,8.569,149.540
C08739=1120.357,138.686,-60.113,-179.596,8.565,149.539
C08740=1120.362,138.437,-60.092,-179.597,8.562,149.539
C08741=1120.366,138.189,-60.070,-179.599,8.559,149.539
C08742=1120.371,137.939,-60.049,-179.600,8.556,149.538
C08743=1120.376,137.689,-60.028,-179.602,8.552,149.538
C08744=1120.380,137.441,-60.007,-179.604,8.549,149.538
C08745=1120.385,137.192,-59.986,-179.605,8.545,149.537
C08746=1120.391,136.943,-59.965,-179.607,8.542,149.537
C08747=1120.395,136.694,-59.944,-179.608,8.539,149.537
C08748=1120.399,136.444,-59.923,-179.610,8.535,149.536
C08749=1120.404,136.195,-59.902,-179.612,8.532,149.536
C08750=1120.409,135.947,-59.881,-179.613,8.529,149.536
C08751=1120.414,135.697,-59.860,-179.615,8.525,149.536
C08752=1120.418,135.449,-59.839,-179.617,8.523,149.535
C08753=1120.423,135.199,-59.818,-179.618,8.519,149.535
C08754=1120.428,134.950,-59.796,-179.620,8.515,149.535
C08755=1120.432,134.701,-59.776,-179.622,8.513,149.534
C08756=1120.437,134.452,-59.755,-179.623,8.509,149.534
C08757=1120.442,134.203,-59.735,-179.625,8.506,149.534
C08758=1120.447,133.953,-59.714,-179.627,8.502,149.534
C08759=1120.451,133.705,-59.693,-179.629,8.499,149.533
C08760=1120.456,133.456,-59.672,-179.630,8.496,149.533
C08761=1120.461,133.207,-59.651,-179.632,8.492,149.533
C08762=1120.465,132.957,-59.630,-179.634,8.489,149.532
C08763=1120.470,132.708,-59.610,-179.635,8.486,149.532
C08764=1120.475,132.459,-59.589,-179.637,8.482,149.532
C08765=1120.479,132.210,-59.567,-179.638,8.479,149.531
C08766=1120.484,131.961,-59.547,-179.640,8.476,149.531
C08767=1120.489,131.712,-59.526,-179.642,8.472,149.531
C08768=1120.494,131.463,-59.505,-179.644,8.470,149.531
C08769=1120.497,131.248,-59.487,-179.645,8.466,149.530
C08770=1120.502,131.035,-59.470,-179.647,8.463,149.530
C08771=1120.506,130.820,-59.452,-179.648,8.460,149.530
C08772=1120.510,130.606,-59.434,-179.650,8.457,149.530
C08773=1120.514,130.392,-59.416,-179.651,8.455,149.529
C08774=1120.518,130.178,-59.399,-179.653,8.452,149.529
C08775=1120.523,129.963,-59.381,-179.654,8.449,149.529
C08776=1120.527,129.749,-59.363,-179.655,8.447,149.529
C08777=1120.531,129.500,-59.342,-179.657,8.443,149.528
C08778=1120.536,129.250,-59.322,-179.659,8.439,149.528
C08779=1120.540,129.001,-59.301,-179.661,8.437,149.528
C08780=1120.545,128.752,-59.281,-179.663,8.433,149.527
C08781=1120.550,128.503,-59.260,-179.664,8.429,149.527
C08782=1120.554,128.254,-59.239,-179.666,8.426,149.527
C08783=1120.560,128.005,-59.218,-179.668,8.423,149.527
C08784=1120.564,127.756,-59.198,-179.670,8.419,149.526
C08785=1120.568,127.507,-59.178,-179.671,8.416,149.526
C08786=1120.574,127.258,-59.157,-179.673,8.413,149.526
C08787=1120.578,127.009,-59.136,-179.675,8.409,149.525
C08788=1120.582,126.760,-59.116,-179.676,8.407,149.525
C08789=1120.588,126.511,-59.095,-179.678,8.403,149.525
C08790=1120.592,126.262,-59.075,-179.680,8.399,149.525
C08791=1120.597,126.012,-59.055,-179.682,8.397,149.524
C08792=1120.602,125.763,-59.034,-179.684,8.393,149.524
C08793=1120.607,125.515,-59.014,-179.685,8.389,149.524
C08794=1120.611,125.266,-58.994,-179.687,8.387,149.523
C08795=1120.617,125.016,-58.973,-179.689,8.383,149.523
C08796=1120.621,124.767,-58.952,-179.691,8.380,149.523
C08797=1120.626,124.518,-58.933,-179.693,8.376,149.523
C08798=1120.630,124.269,-58.912,-179.694,8.373,149.522
C08799=1120.635,124.020,-58.891,-179.696,8.369,149.522
C08800=1120.640,123.771,-58.871,-179.698,8.366,149.522
C08801=1120.645,123.521,-58.851,-179.700,8.363,149.522
C08802=1120.649,123.272,-58.831,-179.701,8.359,149.521
C08803=1120.654,123.023,-58.810,-179.703,8.356,149.521
C08804=1120.659,122.774,-58.790,-179.705,8.352,149.521
C08805=1120.663,122.524,-58.770,-179.707,8.350,149.521
C08806=1120.668,122.275,-58.750,-179.709,8.346,149.520
C08807=1120.672,122.027,-58.729,-179.710,8.342,149.520
C08808=1120.678,121.777,-58.709,-179.712,8.340,149.520
C08809=1120.683,121.528,-58.689,-179.714,8.336,149.519
C08810=1120.687,121.279,-58.669,-179.716,8.333,149.519
C08811=1120.692,121.030,-58.649,-179.718,8.329,149.519
C08812=1120.696,120.781,-58.629,-179.719,8.326,149.519
C08813=1120.701,120.532,-58.608,-179.721,8.322,149.518
C08814=1120.706,120.282,-58.588,-179.723,8.319,149.518
C08815=1120.711,120.033,-58.568,-179.725,8.315,149.518
C08816=1120.716,119.784,-58.548,-179.726,8.312,149.518
C08817=1120.721,119.535,-58.528,-179.728,8.309,149.517
C08818=1120.725,119.286,-58.508,-179.730,8.305,149.517
C08819=1120.730,119.037,-58.488,-179.732,8.302,149.517
C08820=1120.734,118.788,-58.467,-179.734,8.298,149.516
C08821=1120.739,118.538,-58.448,-179.735,8.295,149.516
C08822=1120.744,118.290,-58.428,-179.738,8.292,149.516
C08823=1120.749,118.040,-58.408,-179.740,8.288,149.516
C08824=1120.754,117.791,-58.387,-179.742,8.285,149.515
C08825=1120.758,117.577,-58.371,-179.743,8.282,149.515
C08826=1120.761,117.363,-58.353,-179.744,8.279,149.515
C08827=1120.766,117.148,-58.337,-179.746,8.276,149.515
C08828=1120.770,116.934,-58.319,-179.748,8.273,149.514
C08829=1120.774,116.719,-58.302,-179.749,8.270,149.514
C08830=1120.778,116.506,-58.285,-179.750,8.267,149.514
C08831=1120.782,116.290,-58.268,-179.753,8.264,149.514
C08832=1120.787,116.077,-58.250,-179.754,8.261,149.514
C08833=1120.791,115.827,-58.231,-179.756,8.258,149.513
C08834=1120.797,115.578,-58.211,-179.757,8.255,149.513
C08835=1120.801,115.329,-58.191,-179.759,8.251,149.513
C08836=1120.806,115.080,-58.171,-179.761,8.247,149.512
C08837=1120.810,114.831,-58.151,-179.763,8.244,149.512
C08838=1120.816,114.582,-58.132,-179.765,8.240,149.512
C08839=1120.820,114.332,-58.112,-179.767,8.237,149.512
C08840=1120.825,114.083,-58.092,-179.769,8.233,149.511
C08841=1120.830,113.834,-58.072,-179.770,8.230,149.511
C08842=1120.835,113.585,-58.053,-179.772,8.227,149.511
C08843=1120.839,113.336,-58.034,-179.774,8.223,149.510
C08844=1120.843,113.087,-58.013,-179.776,8.220,149.510
C08845=1120.848,112.837,-57.994,-179.778,8.216,149.510
C08846=1120.853,112.588,-57.974,-179.780,8.213,149.510
C08847=1120.858,112.339,-57.955,-179.782,8.209,149.509
C08848=1120.863,112.090,-57.934,-179.783,8.206,149.509
C08849=1120.868,111.841,-57.915,-179.785,8.202,149.509
C08850=1120.873,111.591,-57.895,-179.787,8.199,149.508
C08851=1120.877,111.342,-57.876,-179.789,8.195,149.508
C08852=1120.883,111.093,-57.856,-179.791,8.192,149.508
C08853=1120.886,110.844,-57.837,-179.793,8.188,149.508
C08854=1120.891,110.595,-57.817,-179.795,8.185,149.508
C08855=1120.897,110.346,-57.798,-179.798,8.180,149.507
C08856=1120.901,110.096,-57.778,-179.800,8.177,149.507
C08857=1120.906,109.847,-57.758,-179.803,8.172,149.507
C08858=1120.911,109.598,-57.739,-179.805,8.169,149.507
C08859=1120.915,109.349,-57.720,-179.807,8.165,149.506
C08860=1120.921,109.100,-57.701,-179.809,8.161,149.506
C08861=1120.925,108.850,-57.681,-179.811,8.157,149.506
C08862=1120.930,108.601,-57.661,-179.814,8.153,149.506
C08863=1120.934,108.353,-57.642,-179.816,8.150,149.505
C08864=1120.939,108.103,-57.622,-179.818,8.146,149.505
C08865=1120.944,107.853,-57.603,-179.821,8.142,149.505
C08866=1120.949,107.605,-57.583,-179.823,8.138,149.505
C08867=1120.953,107.355,-57.564,-179.824,8.134,149.504
C08868=1120.959,107.106,-57.545,-179.827,8.130,149.504
C08869=1120.963,106.857,-57.525,-179.829,8.127,149.504
C08870=1120.969,106.607,-57.507,-179.831,8.123,149.504
C08871=1120.973,106.358,-57.488,-179.833,8.118,149.503
C08872=1120.978,106.109,-57.468,-179.835,8.115,149.503
C08873=1120.983,105.860,-57.449,-179.837,8.111,149.503
C08874=1120.987,105.610,-57.430,-179.839,8.108,149.502
C08875=1120.992,105.362,-57.410,-179.842,8.103,149.502
C08876=1120.997,105.112,-57.391,-179.844,8.100,149.502
C08877=1121.002,104.863,-57.372,-179.845,8.096,149.501
C08878=1121.007,104.614,-57.352,-179.848,8.092,149.501
C08879=1121.012,104.365,-57.334,-179.850,8.088,149.501
C08880=1121.016,104.115,-57.315,-179.852,8.084,149.501
C08881=1121.021,103.901,-57.298,-179.854,8.081,149.500
C08882=1121.025,103.687,-57.282,-179.855,8.078,149.500
C08883=1121.029,103.472,-57.265,-179.857,8.074,149.500
C08884=1121.033,103.258,-57.249,-179.859,8.071,149.499
C08885=1121.037,103.043,-57.232,-179.860,8.068,149.499
C08886=1121.041,102.829,-57.216,-179.862,8.064,149.499
C08887=1121.045,102.614,-57.199,-179.864,8.060,149.499
C08888=1121.049,102.400,-57.184,-179.865,8.058,149.498
C08889=1121.055,102.151,-57.165,-179.867,8.054,149.498
C08890=1121.059,101.902,-57.146,-179.870,8.050,149.498
C08891=1121.064,101.653,-57.126,-179.871,8.046,149.497
C08892=1121.068,101.403,-57.108,-179.873,8.042,149.497
C08893=1121.074,101.154,-57.089,-179.875,8.038,149.497
C08894=1121.078,100.905,-57.070,-179.876,8.034,149.496
C08895=1121.083,100.655,-57.051,-179.879,8.030,149.496
C08896=1121.087,100.406,-57.032,-179.881,8.026,149.496
C08897=1121.093,100.157,-57.013,-179.882,8.022,149.495
C08898=1121.098,99.908,-56.995,-179.884,8.019,149.495
C08899=1121.102,99.658,-56.975,-179.886,8.015,149.494
C08900=1121.107,99.409,-56.957,-179.888,8.011,149.494
C08901=1121.112,99.160,-56.937,-179.890,8.007,149.494
C08902=1121.117,98.910,-56.919,-179.892,8.003,149.493
C08903=1121.122,98.662,-56.900,-179.894,7.999,149.493
C08904=1121.127,98.412,-56.882,-179.895,7.995,149.492
C08905=1121.131,98.163,-56.863,-179.897,7.992,149.492
C08906=1121.136,97.914,-56.843,-179.899,7.988,149.492
C08907=1121.141,97.664,-56.825,-179.900,7.984,149.491
C08908=1121.146,97.416,-56.806,-179.902,7.980,149.491
C08909=1121.151,97.166,-56.788,-179.904,7.976,149.491
C08910=1121.156,96.917,-56.770,-179.905,7.972,149.490
C08911=1121.161,96.668,-56.751,-179.908,7.968,149.490
C08912=1121.165,96.418,-56.732,-179.909,7.964,149.489
C08913=1121.170,96.169,-56.714,-179.911,7.960,149.489
C08914=1121.175,95.920,-56.695,-179.913,7.956,149.489
C08915=1121.179,95.670,-56.676,-179.914,7.952,149.488
C08916=1121.184,95.421,-56.658,-179.916,7.948,149.488
C08917=1121.190,95.172,-56.639,-179.917,7.945,149.487
C08918=1121.194,94.923,-56.620,-179.919,7.941,149.487
C08919=1121.199,94.673,-56.602,-179.921,7.937,149.486
C08920=1121.205,94.424,-56.584,-179.922,7.933,149.486
C08921=1121.209,94.175,-56.565,-179.924,7.929,149.486
C08922=1121.213,93.925,-56.547,-179.925,7.925,149.485
C08923=1121.219,93.676,-56.528,-179.927,7.921,149.485
C08924=1121.224,93.427,-56.509,-179.929,7.917,149.484
C08925=1121.228,93.178,-56.491,-179.930,7.913,149.484
C08926=1121.233,92.928,-56.473,-179.932,7.910,149.483
C08927=1121.238,92.680,-56.454,-179.933,7.906,149.483
C08928=1121.243,92.430,-56.435,-179.935,7.902,149.483
C08929=1121.248,92.180,-56.417,-179.937,7.898,149.482
C08930=1121.252,91.931,-56.399,-179.938,7.894,149.482
C08931=1121.257,91.683,-56.381,-179.940,7.890,149.481
C08932=1121.262,91.433,-56.362,-179.941,7.887,149.481
C08933=1121.267,91.183,-56.344,-179.942,7.883,149.480
C08934=1121.272,90.934,-56.326,-179.944,7.879,149.480
C08935=1121.277,90.685,-56.308,-179.945,7.875,149.479
C08936=1121.282,90.436,-56.290,-179.947,7.871,149.479
C08937=1121.286,90.221,-56.273,-179.948,7.868,149.479
C08938=1121.290,90.007,-56.258,-179.949,7.864,149.478
C08939=1121.294,89.793,-56.242,-179.950,7.861,149.478
C08940=1121.298,89.578,-56.226,-179.951,7.858,149.477
C08941=1121.303,89.363,-56.211,-179.953,7.854,149.477
C08942=1121.306,89.149,-56.195,-179.954,7.851,149.477
C08943=1121.310,88.934,-56.179,-179.955,7.848,149.476
C08944=1121.315,88.719,-56.164,-179.957,7.844,149.476
C08945=1121.320,88.470,-56.146,-179.958,7.841,149.475
C08946=1121.325,88.221,-56.128,-179.959,7.837,149.475
C08947=1121.330,87.972,-56.110,-179.961,7.833,149.474
C08948=1121.334,87.722,-56.091,-179.962,7.829,149.474
C08949=1121.339,87.473,-56.073,-179.963,7.825,149.473
C08950=1121.344,87.224,-56.055,-179.964,7.822,149.473
C08951=1121.349,86.974,-56.037,-179.966,7.818,149.472
C08952=1121.354,86.725,-56.019,-179.967,7.814,149.472
C08953=1121.359,86.476,-56.001,-179.969,7.810,149.471
C08954=1121.363,86.226,-55.983,-179.970,7.806,149.471
C08955=1121.368,85.977,-55.965,-179.971,7.803,149.470
C08956=1121.374,85.727,-55.946,-179.972,7.798,149.470
C08957=1121.379,85.478,-55.928,-179.974,7.794,149.469
C08958=1121.384,85.229,-55.910,-179.975,7.791,149.469
C08959=1121.389,84.980,-55.892,-179.976,7.787,149.468
C08960=1121.393,84.731,-55.875,-179.978,7.783,149.468
C08961=1121.398,84.482,-55.857,-179.979,7.779,149.467
C08962=1121.403,84.232,-55.838,-179.980,7.776,149.467
C08963=1121.408,83.983,-55.820,-179.981,7.772,149.466
C08964=1121.412,83.733,-55.802,-179.982,7.767,149.466
C08965=1121.417,83.484,-55.784,-179.983,7.764,149.465
C08966=1121.422,83.235,-55.767,-179.984,7.760,149.465
C08967=1121.427,82.986,-55.750,-179.986,7.756,149.464
C08968=1121.432,82.736,-55.732,-179.987,7.753,149.464
C08969=1121.437,82.487,-55.714,-179.988,7.749,149.463
C08970=1121.442,82.238,-55.696,-179.990,7.745,149.463
C08971=1121.446,81.989,-55.678,-179.990,7.741,149.462
C08972=1121.451,81.740,-55.660,-179.992,7.738,149.462
C08973=1121.457,81.490,-55.642,-179.992,7.734,149.461
C08974=1121.461,81.240,-55.624,-179.994,7.730,149.460
C08975=1121.466,80.991,-55.606,-179.994,7.727,149.460
C08976=1121.471,80.742,-55.588,-179.996,7.723,149.459
C08977=1121.476,80.492,-55.571,-179.997,7.718,149.459
C08978=1121.481,80.243,-55.553,-179.998,7.715,149.458
C08979=1121.485,79.994,-55.535,-179.999,7.711,149.458
C08980=1121.490,79.745,-55.518,180.000,7.708,149.457
C08981=1121.495,79.495,-55.500,179.999,7.704,149.457
C08982=1121.500,79.246,-55.482,179.998,7.701,149.456
C08983=1121.505,78.996,-55.464,179.997,7.696,149.456
C08984=1121.510,78.747,-55.447,179.996,7.693,149.455
C08985=1121.515,78.497,-55.429,179.995,7.689,149.454
C08986=1121.519,78.249,-55.412,179.994,7.685,149.454
C08987=1121.524,77.999,-55.394,179.992,7.681,149.453
C08988=1121.529,77.750,-55.376,179.992,7.678,149.453
C08989=1121.534,77.500,-55.358,179.990,7.674,149.452
C08990=1121.540,77.251,-55.341,179.990,7.671,149.452
C08991=1121.544,77.001,-55.323,179.989,7.667,149.451
C08992=1121.549,76.753,-55.306,179.988,7.663,149.451
C08993=1121.553,76.538,-55.290,179.987,7.660,149.450
C08994=1121.558,76.323,-55.276,179.985,7.656,149.450
C08995=1121.562,76.109,-55.261,179.984,7.653,149.449
C08996=1121.566,75.894,-55.245,179.983,7.649,149.449
C08997=1121.570,75.679,-55.230,179.982,7.646,149.448
C08998=1121.574,75.465,-55.216,179.981,7.643,149.448
C08999=1121.578,75.251,-55.200,179.979,7.639,149.448
C09000=1121.583,75.035,-55.185,179.978,7.636,149.447
C09001=1121.588,74.786,-55.168,179.977,7.632,149.447
C09002=1121.593,74.536,-55.150,179.975,7.628,149.446
C09003=1121.597,74.287,-55.133,179.974,7.624,149.446
C09004=1121.603,74.038,-55.116,179.972,7.620,149.445
C09005=1121.608,73.789,-55.098,179.971,7.616,149.445
C09006=1121.612,73.540,-55.081,179.969,7.612,149.444
C09007=1121.617,73.291,-55.063,179.968,7.608,149.444
C09008=1121.622,73.041,-55.046,179.967,7.604,149.443
C09009=1121.627,72.792,-55.029,179.965,7.600,149.443
C09010=1121.632,72.542,-55.011,179.963,7.596,149.442
C09011=1121.637,72.293,-54.993,179.962,7.592,149.442
C09012=1121.641,72.043,-54.977,179.961,7.588,149.441
C09013=1121.646,71.794,-54.960,179.959,7.584,149.441
C09014=1121.652,71.545,-54.942,179.958,7.581,149.440
C09015=1121.656,71.296,-54.925,179.957,7.577,149.440
C09016=1121.661,71.047,-54.907,179.955,7.573,149.439
C09017=1121.666,70.797,-54.890,179.954,7.569,149.439
C09018=1121.671,70.547,-54.873,179.952,7.565,149.439
C09019=1121.676,70.298,-54.855,179.951,7.561,149.438
C09020=1121.680,70.049,-54.839,179.950,7.557,149.437
C09021=1121.686,69.799,-54.822,179.948,7.553,149.437
C09022=1121.691,69.550,-54.804,179.947,7.548,149.436
C09023=1121.696,69.301,-54.787,179.945,7.545,149.436
C09024=1121.701,69.051,-54.770,179.944,7.541,149.436
C09025=1121.705,68.802,-54.753,179.942,7.537,149.435
C09026=1121.710,68.552,-54.735,179.941,7.532,149.434
C09027=1121.715,68.304,-54.719,179.940,7.529,149.434
C09028=1121.720,68.054,-54.702,179.938,7.525,149.434
C09029=1121.725,67.804,-54.685,179.937,7.520,149.433
C09030=1121.730,67.555,-54.667,179.936,7.517,149.433
C09031=1121.734,67.306,-54.650,179.934,7.513,149.432
C09032=1121.740,67.057,-54.633,179.933,7.509,149.431
C09033=1121.745,66.807,-54.617,179.932,7.505,149.431
C09034=1121.750,66.557,-54.599,179.930,7.501,149.431
C09035=1121.754,66.308,-54.582,179.929,7.497,149.430
C09036=1121.760,66.059,-54.565,179.927,7.493,149.430
C09037=1121.764,65.810,-54.549,179.926,7.489,149.429
C09038=1121.770,65.560,-54.531,179.925,7.485,149.428
C09039=1121.774,65.311,-54.515,179.923,7.481,149.428
C09040=1121.779,65.061,-54.497,179.922,7.477,149.428
C09041=1121.784,64.812,-54.481,179.920,7.473,149.427
C09042=1121.790,64.562,-54.464,179.919,7.469,149.427
C09043=1121.794,64.313,-54.447,179.917,7.465,149.426
C09044=1121.799,64.065,-54.430,179.916,7.461,149.425
C09045=1121.804,63.815,-54.413,179.915,7.458,149.425
C09046=1121.809,63.565,-54.396,179.914,7.454,149.425
C09047=1121.814,63.315,-54.379,179.913,7.449,149.424
C09048=1121.819,63.067,-54.363,179.911,7.445,149.424
C09049=1121.822,62.852,-54.349,179.910,7.442,149.423
C09050=1121.828,62.637,-54.334,179.909,7.438,149.423
C09051=1121.832,62.422,-54.319,179.908,7.435,149.422
C09052=1121.835,62.207,-54.305,179.906,7.431,149.422
C09053=1121.840,61.993,-54.290,179.905,7.428,149.421
C09054=1121.844,61.778,-54.276,179.904,7.424,149.421
C09055=1121.849,61.564,-54.261,179.903,7.421,149.421
C09056=1121.853,61.348,-54.247,179.902,7.418,149.420
C09057=1121.858,61.100,-54.231,179.901,7.414,149.419
C09058=1121.863,60.850,-54.214,179.899,7.410,149.419
C09059=1121.867,60.600,-54.197,179.898,7.406,149.418
C09060=1121.872,60.352,-54.181,179.896,7.402,149.418
C09061=1121.878,60.102,-54.163,179.895,7.398,149.418
C09062=1121.882,59.852,-54.148,179.894,7.393,149.417
C09063=1121.887,59.603,-54.131,179.892,7.390,149.416
C09064=1121.892,59.353,-54.115,179.891,7.385,149.416
C09065=1121.897,59.104,-54.097,179.889,7.381,149.415
C09066=1121.902,58.855,-54.081,179.888,7.377,149.415
C09067=1121.907,58.605,-54.064,179.887,7.373,149.414
C09068=1121.912,58.357,-54.048,179.886,7.370,149.414
C09069=1121.917,58.106,-54.031,179.885,7.366,149.413
C09070=1121.922,57.857,-54.015,179.883,7.362,149.413
C09071=1121.927,57.608,-53.998,179.882,7.358,149.412
C09072=1121.931,57.358,-53.982,179.881,7.354,149.412
C09073=1121.937,57.109,-53.966,179.879,7.349,149.411
C09074=1121.942,56.859,-53.949,179.878,7.345,149.411
C09075=1121.946,56.610,-53.932,179.876,7.342,149.410
C09076=1121.952,56.361,-53.916,179.875,7.337,149.410
C09077=1121.956,56.111,-53.900,179.874,7.333,149.409
C09078=1121.962,55.862,-53.883,179.873,7.329,149.408
C09079=1121.967,55.612,-53.866,179.871,7.325,149.408
C09080=1121.972,55.364,-53.850,179.870,7.321,149.407
C09081=1121.976,55.113,-53.834,179.869,7.318,149.407
C09082=1121.981,54.864,-53.818,179.868,7.313,149.406
C09083=1121.986,54.615,-53.801,179.866,7.309,149.406
C09084=1121.991,54.365,-53.785,179.865,7.305,149.405
C09085=1121.997,54.116,-53.768,179.864,7.301,149.405
C09086=1122.001,53.866,-53.752,179.863,7.297,149.404
C09087=1122.007,53.617,-53.736,179.861,7.293,149.404
C09088=1122.011,53.368,-53.719,179.860,7.289,149.403
C09089=1122.016,53.118,-53.704,179.858,7.285,149.403
C09090=1122.021,52.869,-53.687,179.857,7.281,149.402
C09091=1122.026,52.619,-53.672,179.856,7.277,149.402
C09092=1122.031,52.370,-53.655,179.855,7.272,149.401
C09093=1122.036,52.121,-53.639,179.853,7.268,149.401
C09094=1122.041,51.871,-53.623,179.853,7.265,149.400
C09095=1122.046,51.622,-53.606,179.851,7.261,149.399
C09096=1122.051,51.372,-53.590,179.850,7.257,149.399
C09097=1122.056,51.123,-53.574,179.848,7.253,149.398
C09098=1122.061,50.873,-53.558,179.847,7.248,149.398
C09099=1122.066,50.624,-53.541,179.846,7.244,149.397
C09100=1122.072,50.375,-53.526,179.845,7.240,149.397
C09101=1122.076,50.125,-53.509,179.844,7.236,149.396
C09102=1122.081,49.876,-53.493,179.842,7.232,149.396
C09103=1122.086,49.626,-53.477,179.841,7.228,149.395
C09104=1122.091,49.377,-53.461,179.839,7.224,149.394
C09105=1122.095,49.162,-53.447,179.839,7.220,149.394
C09106=1122.100,48.947,-53.434,179.837,7.216,149.393
C09107=1122.104,48.733,-53.420,179.836,7.213,149.393
C09108=1122.108,48.518,-53.406,179.836,7.210,149.393
C09109=1122.112,48.303,-53.393,179.834,7.206,149.392
C09110=1122.117,48.088,-53.379,179.834,7.203,149.391
C09111=1122.121,47.873,-53.365,179.833,7.200,149.391
C09112=1122.125,47.659,-53.351,179.831,7.196,149.391
C09113=1122.130,47.408,-53.335,179.830,7.191,149.390
C09114=1122.135,47.160,-53.319,179.829,7.187,149.389
C09115=1122.140,46.910,-53.303,179.827,7.183,149.389
C09116=1122.145,46.660,-53.287,179.826,7.179,149.388
C09117=1122.150,46.412,-53.272,179.825,7.175,149.388
C09118=1122.154,46.162,-53.256,179.824,7.171,149.387
C09119=1122.160,45.912,-53.240,179.823,7.167,149.387
C09120=1122.165,45.663,-53.225,179.822,7.163,149.386
C09121=1122.170,45.413,-53.208,179.821,7.159,149.385
C09122=1122.175,45.164,-53.192,179.819,7.155,149.385
C09123=1122.180,44.915,-53.177,179.818,7.151,149.384
C09124=1122.185,44.664,-53.161,179.817,7.146,149.384
C09125=1122.189,44.416,-53.145,179.816,7.142,149.383
C09126=1122.195,44.167,-53.130,179.814,7.138,149.383
C09127=1122.200,43.916,-53.114,179.813,7.134,149.382
C09128=1122.205,43.667,-53.098,179.812,7.130,149.381
